LIN {X 0,Y 305.453,Z 160.427,A -85,B 0,C 180,E1 -15811.108,E2 -15811.108} C_VEL
LIN {X 0,Y 305.478,Z 160.428,A -85,B 0,C 180,E1 -15814.08,E2 -15814.08} C_VEL
LIN {X 0,Y 305.457,Z 160.438,A -85,B 0,C 180,E1 -15818.4,E2 -15818.4} C_VEL
LIN {X 0,Y 305.499,Z 160.427,A -85,B 0,C 180,E1 -15821.213,E2 -15821.213} C_VEL
LIN {X 0,Y 305.569,Z 160.419,A -85,B 0,C 180,E1 -15825.346,E2 -15825.346} C_VEL
LIN {X 0,Y 305.622,Z 160.412,A -85,B 0,C 180,E1 -15829.4,E2 -15829.4} C_VEL
LIN {X 0,Y 305.753,Z 160.399,A -85,B 0,C 180,E1 -15832.074,E2 -15832.074} C_VEL
LIN {X 0,Y 305.659,Z 160.409,A -85,B 0,C 180,E1 -15834.724,E2 -15834.724} C_VEL
LIN {X 0,Y 305.938,Z 160.372,A -85,B 0,C 180,E1 -15838.684,E2 -15838.684} C_VEL
LIN {X 0,Y 305.939,Z 160.373,A -85,B 0,C 180,E1 -15841.317,E2 -15841.317} C_VEL
LIN {X 0,Y 305.788,Z 160.391,A -85,B 0,C 180,E1 -15846.599,E2 -15846.599} C_VEL
LIN {X 0,Y 305.699,Z 160.403,A -85,B 0,C 180,E1 -15849.262,E2 -15849.262} C_VEL
LIN {X 0,Y 305.576,Z 160.422,A -85,B 0,C 180,E1 -15853.297,E2 -15853.297} C_VEL
LIN {X 0,Y 305.518,Z 160.424,A -85,B 0,C 180,E1 -15856.025,E2 -15856.025} C_VEL
LIN {X 0,Y 305.483,Z 160.43,A -85,B 0,C 180,E1 -15860.188,E2 -15860.188} C_VEL
LIN {X 0,Y 305.491,Z 160.432,A -85,B 0,C 180,E1 -15863.04,E2 -15863.04} C_VEL
LIN {X 0,Y 305.472,Z 160.431,A -85,B 0,C 180,E1 -15866.197,E2 -15866.197} C_VEL
LIN {X 0,Y 305.451,Z 160.438,A -85,B 0,C 180,E1 -15869.033,E2 -15869.033} C_VEL
LIN {X 0,Y 305.44,Z 160.435,A -85,B 0,C 180,E1 -15871.953,E2 -15871.953} C_VEL
LIN {X 0,Y 305.466,Z 160.436,A -85,B 0,C 180,E1 -15875.114,E2 -15875.114} C_VEL
LIN {X 0,Y 305.437,Z 160.438,A -85,B 0,C 180,E1 -15878.525,E2 -15878.525} C_VEL
LIN {X 0,Y 305.439,Z 160.44,A -85,B 0,C 180,E1 -15882.582,E2 -15882.582} C_VEL
LIN {X 0,Y 305.424,Z 160.441,A -85,B 0,C 180,E1 -15886.344,E2 -15886.344} C_VEL
LIN {X 0,Y 305.414,Z 160.44,A -85,B 0,C 180,E1 -15889.885,E2 -15889.885} C_VEL
LIN {X 0,Y 305.467,Z 160.433,A -85,B 0,C 180,E1 -15893.636,E2 -15893.636} C_VEL
LIN {X 0,Y 305.469,Z 160.437,A -85,B 0,C 180,E1 -15896.483,E2 -15896.483} C_VEL
LIN {X 0,Y 305.467,Z 160.528,A -85,B 0,C 180,E1 -15898.422,E2 -15898.422} C_VEL
LIN {X 0,Y 307.798,Z 171.715,A -85,B 0,C 180,E1 -15901.719,E2 -15901.719} C_VEL
LIN {X 0,Y 309.263,Z 179.963,A -85,B 0,C 180,E1 -15904.058,E2 -15904.058} C_VEL
LIN {X 0,Y 308.728,Z 185.546,A -85,B 0,C 180,E1 -15905.524,E2 -15905.524} C_VEL
LIN {X 0,Y 314.413,Z 227.443,A -85,B 0,C 180,E1 -15906.914,E2 -15906.914} C_VEL
LIN {X 0,Y 312.89,Z 293.878,A -85,B 0,C 180,E1 -15908.462,E2 -15908.462} C_VEL
LIN {X 0,Y 312.195,Z 307.17,A -85,B 0,C 180,E1 -15909.018,E2 -15909.018} C_VEL
LIN {X 0,Y 311.167,Z 320.508,A -85,B 0,C 180,E1 -15909.852,E2 -15909.852} C_VEL
LIN {X 0,Y 310.022,Z 331.7,A -85,B 0,C 180,E1 -15910.809,E2 -15910.809} C_VEL
LIN {X 0,Y 308.738,Z 343.365,A -85,B 0,C 180,E1 -15912.102,E2 -15912.102} C_VEL
LIN {X 0,Y 307.518,Z 354.294,A -85,B 0,C 180,E1 -15913.638,E2 -15913.638} C_VEL
LIN {X 0,Y 306.372,Z 364.129,A -85,B 0,C 180,E1 -15915.384,E2 -15915.384} C_VEL
LIN {X 0,Y 305.291,Z 373.098,A -85,B 0,C 180,E1 -15917.367,E2 -15917.367} C_VEL
LIN {X 0,Y 304.512,Z 380.276,A -85,B 0,C 180,E1 -15919.36,E2 -15919.36} C_VEL
LIN {X 0,Y 304.015,Z 385.985,A -85,B 0,C 180,E1 -15921.358,E2 -15921.358} C_VEL
LIN {X 0,Y 303.748,Z 390.465,A -85,B 0,C 180,E1 -15923.356,E2 -15923.356} C_VEL
LIN {X 0,Y 303.669,Z 392.822,A -85,B 0,C 180,E1 -15924.688,E2 -15924.688} C_VEL
LIN {X 0,Y 303.664,Z 394.742,A -85,B 0,C 180,E1 -15926.018,E2 -15926.018} C_VEL
LIN {X 0,Y 303.642,Z 396.207,A -85,B 0,C 180,E1 -15927.346,E2 -15927.346} C_VEL
LIN {X 0,Y 303.634,Z 397.229,A -85,B 0,C 180,E1 -15928.673,E2 -15928.673} C_VEL
LIN {X 0,Y 303.671,Z 397.858,A -85,B 0,C 180,E1 -15930,E2 -15930} C_VEL
LIN {X 0,Y 303.608,Z 398.092,A -85,B 0,C 180,E1 -15931.326,E2 -15931.326} C_VEL
LIN {X 0,Y 303.622,Z 397.918,A -85,B 0,C 180,E1 -15932.653,E2 -15932.653} C_VEL
LIN {X 0,Y 303.624,Z 397.32,A -85,B 0,C 180,E1 -15933.982,E2 -15933.982} C_VEL
LIN {X 0,Y 303.732,Z 394.961,A -85,B 0,C 180,E1 -15936.643,E2 -15936.643} C_VEL
LIN {X 0,Y 304.114,Z 392.081,A -85,B 0,C 180,E1 -15938.639,E2 -15938.639} C_VEL
LIN {X 0,Y 304.723,Z 388.193,A -85,B 0,C 180,E1 -15940.632,E2 -15940.632} C_VEL
LIN {X 0,Y 305.625,Z 383.199,A -85,B 0,C 180,E1 -15942.618,E2 -15942.618} C_VEL
LIN {X 0,Y 307.01,Z 376.951,A -85,B 0,C 180,E1 -15944.584,E2 -15944.584} C_VEL
LIN {X 0,Y 308.52,Z 369.636,A -85,B 0,C 180,E1 -15946.439,E2 -15946.439} C_VEL
LIN {X 0,Y 310.07,Z 361.462,A -85,B 0,C 180,E1 -15948.125,E2 -15948.125} C_VEL
LIN {X 0,Y 312.018,Z 351.681,A -85,B 0,C 180,E1 -15949.747,E2 -15949.747} C_VEL
LIN {X 0,Y 313.987,Z 341.067,A -85,B 0,C 180,E1 -15951.157,E2 -15951.157} C_VEL
LIN {X 0,Y 315.629,Z 330.837,A -85,B 0,C 180,E1 -15952.243,E2 -15952.243} C_VEL
LIN {X 0,Y 317.331,Z 318.676,A -85,B 0,C 180,E1 -15953.235,E2 -15953.235} C_VEL
LIN {X 0,Y 318.848,Z 305.214,A -85,B 0,C 180,E1 -15954.022,E2 -15954.022} C_VEL
LIN {X 0,Y 319.839,Z 292.7,A -85,B 0,C 180,E1 -15954.504,E2 -15954.504} C_VEL
LIN {X 0,Y 321.622,Z 229.197,A -85,B 0,C 180,E1 -15956.002,E2 -15956.002} C_VEL
LIN {X 0,Y 318.654,Z 211.067,A -85,B 0,C 180,E1 -15956.804,E2 -15956.804} C_VEL
LIN {X 0,Y 314.686,Z 192.542,A -85,B 0,C 180,E1 -15957.753,E2 -15957.753} C_VEL
LIN {X 0,Y 311.096,Z 184.219,A -85,B 0,C 180,E1 -15958.444,E2 -15958.444} C_VEL
LIN {X 0,Y 309.125,Z 174.684,A -85,B 0,C 180,E1 -15961.527,E2 -15961.527} C_VEL
LIN {X 0,Y 306.659,Z 164.84,A -85,B 0,C 180,E1 -15964.956,E2 -15964.956} C_VEL
LIN {X 0,Y 305.47,Z 160.428,A -85,B 0,C 180,E1 -15966.618,E2 -15966.618} C_VEL
LIN {X 0,Y 305.412,Z 160.433,A -85,B 0,C 180,E1 -15970.115,E2 -15970.115} C_VEL
LIN {X 0,Y 305.423,Z 160.439,A -85,B 0,C 180,E1 -15973.656,E2 -15973.656} C_VEL
LIN {X 0,Y 305.436,Z 160.439,A -85,B 0,C 180,E1 -15977.418,E2 -15977.418} C_VEL
LIN {X 0,Y 305.462,Z 160.431,A -85,B 0,C 180,E1 -15981.595,E2 -15981.595} C_VEL
LIN {X 0,Y 305.463,Z 160.429,A -85,B 0,C 180,E1 -15984.886,E2 -15984.886} C_VEL
LIN {X 0,Y 305.443,Z 160.432,A -85,B 0,C 180,E1 -15988.358,E2 -15988.358} C_VEL
LIN {X 0,Y 305.476,Z 160.432,A -85,B 0,C 180,E1 -15991.108,E2 -15991.108} C_VEL
LIN {X 0,Y 305.48,Z 160.424,A -85,B 0,C 180,E1 -15994.079,E2 -15994.079} C_VEL
LIN {X 0,Y 305.457,Z 160.427,A -85,B 0,C 180,E1 -15998.399,E2 -15998.399} C_VEL
LIN {X 0,Y 305.503,Z 160.424,A -85,B 0,C 180,E1 -16001.211,E2 -16001.211} C_VEL
LIN {X 0,Y 305.581,Z 160.419,A -85,B 0,C 180,E1 -16005.345,E2 -16005.345} C_VEL
LIN {X 0,Y 305.625,Z 160.414,A -85,B 0,C 180,E1 -16009.399,E2 -16009.399} C_VEL
LIN {X 0,Y 305.748,Z 160.387,A -85,B 0,C 180,E1 -16012.072,E2 -16012.072} C_VEL
LIN {X 0,Y 305.661,Z 160.407,A -85,B 0,C 180,E1 -16014.722,E2 -16014.722} C_VEL
LIN {X 0,Y 305.947,Z 160.372,A -85,B 0,C 180,E1 -16018.683,E2 -16018.683} C_VEL
LIN {X 0,Y 305.942,Z 160.363,A -85,B 0,C 180,E1 -16021.316,E2 -16021.316} C_VEL
LIN {X 0,Y 305.668,Z 160.401,A -85,B 0,C 180,E1 -16025.276,E2 -16025.276} C_VEL
LIN {X 0,Y 305.748,Z 160.4,A -85,B 0,C 180,E1 -16027.927,E2 -16027.927} C_VEL
LIN {X 0,Y 305.601,Z 160.418,A -85,B 0,C 180,E1 -16031.944,E2 -16031.944} C_VEL
LIN {X 0,Y 305.609,Z 160.409,A -85,B 0,C 180,E1 -16035.014,E2 -16035.014} C_VEL
LIN {X 0,Y 305.547,Z 160.423,A -85,B 0,C 180,E1 -16039.428,E2 -16039.428} C_VEL
LIN {X 0,Y 305.486,Z 160.433,A -85,B 0,C 180,E1 -16043.039,E2 -16043.039} C_VEL
LIN {X 0,Y 305.553,Z 160.425,A -85,B 0,C 180,E1 -16046.229,E2 -16046.229} C_VEL
LIN {X 0,Y 305.495,Z 160.434,A -85,B 0,C 180,E1 -16049.049,E2 -16049.049} C_VEL
LIN {X 0,Y 305.443,Z 160.439,A -85,B 0,C 180,E1 -16051.951,E2 -16051.951} C_VEL
LIN {X 0,Y 305.461,Z 160.436,A -85,B 0,C 180,E1 -16055.112,E2 -16055.112} C_VEL
LIN {X 0,Y 305.481,Z 160.531,A -85,B 0,C 180,E1 -16058.995,E2 -16058.995} C_VEL
LIN {X 0,Y 306.938,Z 166.086,A -85,B 0,C 180,E1 -16061.11,E2 -16061.11} C_VEL
LIN {X 0,Y 315.148,Z 182.086,A -85,B 0,C 180,E1 -16062.566,E2 -16062.566} C_VEL
LIN {X 0,Y 322.647,Z 199.055,A -85,B 0,C 180,E1 -16063.867,E2 -16063.867} C_VEL
LIN {X 0,Y 320.218,Z 273.623,A -85,B 0,C 180,E1 -16065.607,E2 -16065.607} C_VEL
LIN {X 0,Y 319.312,Z 286.842,A -85,B 0,C 180,E1 -16066.168,E2 -16066.168} C_VEL
LIN {X 0,Y 318.139,Z 299.763,A -85,B 0,C 180,E1 -16066.995,E2 -16066.995} C_VEL
LIN {X 0,Y 316.565,Z 311.66,A -85,B 0,C 180,E1 -16068.025,E2 -16068.025} C_VEL
LIN {X 0,Y 314.88,Z 322.44,A -85,B 0,C 180,E1 -16069.228,E2 -16069.228} C_VEL
LIN {X 0,Y 313.124,Z 332.579,A -85,B 0,C 180,E1 -16070.649,E2 -16070.649} C_VEL
LIN {X 0,Y 311.124,Z 342.596,A -85,B 0,C 180,E1 -16072.417,E2 -16072.417} C_VEL
LIN {X 0,Y 309.42,Z 350.599,A -85,B 0,C 180,E1 -16074.178,E2 -16074.178} C_VEL
LIN {X 0,Y 307.952,Z 357.327,A -85,B 0,C 180,E1 -16076.004,E2 -16076.004} C_VEL
LIN {X 0,Y 306.491,Z 363.676,A -85,B 0,C 180,E1 -16078.17,E2 -16078.17} C_VEL
LIN {X 0,Y 305.435,Z 368.51,A -85,B 0,C 180,E1 -16080.349,E2 -16080.349} C_VEL
LIN {X 0,Y 304.584,Z 372.051,A -85,B 0,C 180,E1 -16082.517,E2 -16082.517} C_VEL
LIN {X 0,Y 304.096,Z 374.142,A -85,B 0,C 180,E1 -16084.332,E2 -16084.332} C_VEL
LIN {X 0,Y 303.653,Z 375.725,A -85,B 0,C 180,E1 -16086.83,E2 -16086.83} C_VEL
LIN {X 0,Y 303.54,Z 376.02,A -85,B 0,C 180,E1 -16088.256,E2 -16088.256} C_VEL
LIN {X 0,Y 303.461,Z 375.877,A -85,B 0,C 180,E1 -16089.672,E2 -16089.672} C_VEL
LIN {X 0,Y 303.499,Z 374.866,A -85,B 0,C 180,E1 -16091.696,E2 -16091.696} C_VEL
LIN {X 0,Y 303.653,Z 372.729,A -85,B 0,C 180,E1 -16093.875,E2 -16093.875} C_VEL
LIN {X 0,Y 304.054,Z 369.307,A -85,B 0,C 180,E1 -16096.116,E2 -16096.116} C_VEL
LIN {X 0,Y 304.43,Z 365.405,A -85,B 0,C 180,E1 -16098.008,E2 -16098.008} C_VEL
LIN {X 0,Y 305.114,Z 358.942,A -85,B 0,C 180,E1 -16100.387,E2 -16100.387} C_VEL
LIN {X 0,Y 305.975,Z 351.895,A -85,B 0,C 180,E1 -16102.411,E2 -16102.411} C_VEL
LIN {X 0,Y 306.881,Z 344.682,A -85,B 0,C 180,E1 -16104.085,E2 -16104.085} C_VEL
LIN {X 0,Y 308.05,Z 334.951,A -85,B 0,C 180,E1 -16105.912,E2 -16105.912} C_VEL
LIN {X 0,Y 309.279,Z 325.11,A -85,B 0,C 180,E1 -16107.395,E2 -16107.395} C_VEL
LIN {X 0,Y 310.386,Z 314.381,A -85,B 0,C 180,E1 -16108.703,E2 -16108.703} C_VEL
LIN {X 0,Y 311.427,Z 302.397,A -85,B 0,C 180,E1 -16109.839,E2 -16109.839} C_VEL
LIN {X 0,Y 312.319,Z 289.908,A -85,B 0,C 180,E1 -16110.725,E2 -16110.725} C_VEL
LIN {X 0,Y 312.962,Z 277.052,A -85,B 0,C 180,E1 -16111.367,E2 -16111.367} C_VEL
LIN {X 0,Y 313.42,Z 261.752,A -85,B 0,C 180,E1 -16111.807,E2 -16111.807} C_VEL
LIN {X 0,Y 314.938,Z 194.418,A -85,B 0,C 180,E1 -16113.35,E2 -16113.35} C_VEL
LIN {X 0,Y 312.824,Z 183.531,A -85,B 0,C 180,E1 -16113.751,E2 -16113.751} C_VEL
LIN {X 0,Y 308.878,Z 171.653,A -85,B 0,C 180,E1 -16114.305,E2 -16114.305} C_VEL
LIN {X 0,Y 306.47,Z 164.922,A -85,B 0,C 180,E1 -16114.646,E2 -16114.646} C_VEL
LIN {X 0,Y 305.782,Z 160.401,A -85,B 0,C 180,E1 -16116.102,E2 -16116.102} C_VEL
LIN {X 0,Y 305.689,Z 160.407,A -85,B 0,C 180,E1 -16119.261,E2 -16119.261} C_VEL
LIN {X 0,Y 305.549,Z 160.424,A -85,B 0,C 180,E1 -16123.298,E2 -16123.298} C_VEL
LIN {X 0,Y 305.488,Z 160.432,A -85,B 0,C 180,E1 -16126.026,E2 -16126.026} C_VEL
LIN {X 0,Y 305.475,Z 160.435,A -85,B 0,C 180,E1 -16129.393,E2 -16129.393} C_VEL
LIN {X 0,Y 305.452,Z 160.433,A -85,B 0,C 180,E1 -16133.026,E2 -16133.026} C_VEL
LIN {X 0,Y 305.446,Z 160.426,A -85,B 0,C 180,E1 -16136.19,E2 -16136.19} C_VEL
LIN {X 0,Y 305.421,Z 160.437,A -85,B 0,C 180,E1 -16139.026,E2 -16139.026} C_VEL
LIN {X 0,Y 305.433,Z 160.437,A -85,B 0,C 180,E1 -16141.954,E2 -16141.954} C_VEL
LIN {X 0,Y 305.458,Z 160.435,A -85,B 0,C 180,E1 -16145.114,E2 -16145.114} C_VEL
LIN {X 0,Y 305.43,Z 160.436,A -85,B 0,C 180,E1 -16148.525,E2 -16148.525} C_VEL
LIN {X 0,Y 305.432,Z 160.438,A -85,B 0,C 180,E1 -16152.582,E2 -16152.582} C_VEL
LIN {X 0,Y 305.419,Z 160.433,A -85,B 0,C 180,E1 -16156.345,E2 -16156.345} C_VEL
LIN {X 0,Y 305.422,Z 160.432,A -85,B 0,C 180,E1 -16157.218,E2 -16157.218} C_VEL
LIN {X 0,Y 304.785,Z 160.515,A -85,B 0,C 180,E1 -16158.319,E2 -16158.319} C_VEL
LIN {X 0,Y 301.914,Z 160.873,A -85,B 0,C 180,E1 -16160.112,E2 -16160.112} C_VEL
LIN {X 0,Y 299.485,Z 161.177,A -85,B 0,C 180,E1 -16161.566,E2 -16161.566} C_VEL
LIN {X 0,Y 298.479,Z 161.306,A -85,B 0,C 180,E1 -16162.693,E2 -16162.693} C_VEL
LIN {X 0,Y 298.418,Z 161.311,A -85,B 0,C 180,E1 -16163.075,E2 -16163.075} C_VEL
LIN {X 0,Y 298.407,Z 161.309,A -85,B 0,C 180,E1 -16165.582,E2 -16165.582} C_VEL
LIN {X 0,Y 298.372,Z 161.309,A -85,B 0,C 180,E1 -16168.789,E2 -16168.789} C_VEL
LIN {X 0,Y 298.396,Z 161.304,A -85,B 0,C 180,E1 -16171.898,E2 -16171.898} C_VEL
LIN {X 0,Y 298.413,Z 161.311,A -85,B 0,C 180,E1 -16174.918,E2 -16174.918} C_VEL
LIN {X 0,Y 298.39,Z 161.315,A -85,B 0,C 180,E1 -16177.862,E2 -16177.862} C_VEL
LIN {X 0,Y 298.451,Z 161.306,A -85,B 0,C 180,E1 -16180.752,E2 -16180.752} C_VEL
LIN {X 0,Y 298.512,Z 161.298,A -85,B 0,C 180,E1 -16184.991,E2 -16184.991} C_VEL
LIN {X 0,Y 298.58,Z 161.289,A -85,B 0,C 180,E1 -16189.147,E2 -16189.147} C_VEL
LIN {X 0,Y 298.703,Z 161.275,A -85,B 0,C 180,E1 -16191.885,E2 -16191.885} C_VEL
LIN {X 0,Y 298.63,Z 161.285,A -85,B 0,C 180,E1 -16194.599,E2 -16194.599} C_VEL
LIN {X 0,Y 298.905,Z 161.248,A -85,B 0,C 180,E1 -16198.653,E2 -16198.653} C_VEL
LIN {X 0,Y 298.907,Z 161.249,A -85,B 0,C 180,E1 -16201.348,E2 -16201.348} C_VEL
LIN {X 0,Y 298.737,Z 161.269,A -85,B 0,C 180,E1 -16206.756,E2 -16206.756} C_VEL
LIN {X 0,Y 298.63,Z 161.286,A -85,B 0,C 180,E1 -16209.483,E2 -16209.483} C_VEL
LIN {X 0,Y 298.528,Z 161.3,A -85,B 0,C 180,E1 -16213.617,E2 -16213.617} C_VEL
LIN {X 0,Y 298.458,Z 161.302,A -85,B 0,C 180,E1 -16216.414,E2 -16216.414} C_VEL
LIN {X 0,Y 298.447,Z 161.31,A -85,B 0,C 180,E1 -16219.617,E2 -16219.617} C_VEL
LIN {X 0,Y 298.425,Z 161.312,A -85,B 0,C 180,E1 -16223.601,E2 -16223.601} C_VEL
LIN {X 0,Y 298.411,Z 161.312,A -85,B 0,C 180,E1 -16226.583,E2 -16226.583} C_VEL
LIN {X 0,Y 298.397,Z 161.314,A -85,B 0,C 180,E1 -16229.644,E2 -16229.644} C_VEL
LIN {X 0,Y 298.397,Z 161.316,A -85,B 0,C 180,E1 -16232.801,E2 -16232.801} C_VEL
LIN {X 0,Y 298.445,Z 161.311,A -85,B 0,C 180,E1 -16236.806,E2 -16236.806} C_VEL
LIN {X 0,Y 298.352,Z 161.323,A -85,B 0,C 180,E1 -16241.079,E2 -16241.079} C_VEL
LIN {X 0,Y 298.359,Z 161.321,A -85,B 0,C 180,E1 -16245.035,E2 -16245.035} C_VEL
LIN {X 0,Y 298.352,Z 161.322,A -85,B 0,C 180,E1 -16248.921,E2 -16248.921} C_VEL
LIN {X 0,Y 298.402,Z 161.315,A -85,B 0,C 180,E1 -16252.239,E2 -16252.239} C_VEL
LIN {X 0,Y 298.412,Z 161.313,A -85,B 0,C 180,E1 -16255.581,E2 -16255.581} C_VEL
LIN {X 0,Y 298.445,Z 161.51,A -85,B 0,C 180,E1 -16258.108,E2 -16258.108} C_VEL
LIN {X 0,Y 300.709,Z 172.305,A -85,B 0,C 180,E1 -16261.372,E2 -16261.372} C_VEL
LIN {X 0,Y 302.205,Z 180.572,A -85,B 0,C 180,E1 -16263.777,E2 -16263.777} C_VEL
LIN {X 0,Y 301.998,Z 184.584,A -85,B 0,C 180,E1 -16264.868,E2 -16264.868} C_VEL
LIN {X 0,Y 301.902,Z 185.248,A -85,B 0,C 180,E1 -16265.044,E2 -16265.044} C_VEL
LIN {X 0,Y 307.689,Z 228.186,A -85,B 0,C 180,E1 -16266.518,E2 -16266.518} C_VEL
LIN {X 0,Y 306.092,Z 294.136,A -85,B 0,C 180,E1 -16268.092,E2 -16268.092} C_VEL
LIN {X 0,Y 305.32,Z 308.017,A -85,B 0,C 180,E1 -16268.699,E2 -16268.699} C_VEL
LIN {X 0,Y 304.275,Z 321.004,A -85,B 0,C 180,E1 -16269.552,E2 -16269.552} C_VEL
LIN {X 0,Y 302.985,Z 333.629,A -85,B 0,C 180,E1 -16270.698,E2 -16270.698} C_VEL
LIN {X 0,Y 301.565,Z 344.875,A -85,B 0,C 180,E1 -16272.013,E2 -16272.013} C_VEL
LIN {X 0,Y 300.588,Z 354.013,A -85,B 0,C 180,E1 -16273.357,E2 -16273.357} C_VEL
LIN {X 0,Y 299.481,Z 363.35,A -85,B 0,C 180,E1 -16275.04,E2 -16275.04} C_VEL
LIN {X 0,Y 298.328,Z 372.404,A -85,B 0,C 180,E1 -16277.067,E2 -16277.067} C_VEL
LIN {X 0,Y 297.485,Z 379.68,A -85,B 0,C 180,E1 -16279.105,E2 -16279.105} C_VEL
LIN {X 0,Y 296.97,Z 385.468,A -85,B 0,C 180,E1 -16281.151,E2 -16281.151} C_VEL
LIN {X 0,Y 296.69,Z 390.009,A -85,B 0,C 180,E1 -16283.198,E2 -16283.198} C_VEL
LIN {X 0,Y 296.583,Z 392.393,A -85,B 0,C 180,E1 -16284.561,E2 -16284.561} C_VEL
LIN {X 0,Y 296.579,Z 394.34,A -85,B 0,C 180,E1 -16285.923,E2 -16285.923} C_VEL
LIN {X 0,Y 296.567,Z 395.854,A -85,B 0,C 180,E1 -16287.283,E2 -16287.283} C_VEL
LIN {X 0,Y 296.55,Z 396.906,A -85,B 0,C 180,E1 -16288.642,E2 -16288.642} C_VEL
LIN {X 0,Y 296.582,Z 397.56,A -85,B 0,C 180,E1 -16290,E2 -16290} C_VEL
LIN {X 0,Y 296.525,Z 397.819,A -85,B 0,C 180,E1 -16291.358,E2 -16291.358} C_VEL
LIN {X 0,Y 296.546,Z 397.687,A -85,B 0,C 180,E1 -16292.717,E2 -16292.717} C_VEL
LIN {X 0,Y 296.521,Z 397.121,A -85,B 0,C 180,E1 -16294.077,E2 -16294.077} C_VEL
LIN {X 0,Y 296.657,Z 394.812,A -85,B 0,C 180,E1 -16296.803,E2 -16296.803} C_VEL
LIN {X 0,Y 297.066,Z 391.985,A -85,B 0,C 180,E1 -16298.846,E2 -16298.846} C_VEL
LIN {X 0,Y 297.725,Z 388.151,A -85,B 0,C 180,E1 -16300.885,E2 -16300.885} C_VEL
LIN {X 0,Y 298.668,Z 383.216,A -85,B 0,C 180,E1 -16302.917,E2 -16302.917} C_VEL
LIN {X 0,Y 300.147,Z 377.047,A -85,B 0,C 180,E1 -16304.926,E2 -16304.926} C_VEL
LIN {X 0,Y 301.654,Z 370.06,A -85,B 0,C 180,E1 -16306.767,E2 -16306.767} C_VEL
LIN {X 0,Y 303.376,Z 361.636,A -85,B 0,C 180,E1 -16308.574,E2 -16308.574} C_VEL
LIN {X 0,Y 305.38,Z 352.169,A -85,B 0,C 180,E1 -16310.194,E2 -16310.194} C_VEL
LIN {X 0,Y 307.416,Z 341.709,A -85,B 0,C 180,E1 -16311.632,E2 -16311.632} C_VEL
LIN {X 0,Y 309.39,Z 330.102,A -85,B 0,C 180,E1 -16312.893,E2 -16312.893} C_VEL
LIN {X 0,Y 311.158,Z 317.757,A -85,B 0,C 180,E1 -16313.9,E2 -16313.9} C_VEL
LIN {X 0,Y 312.681,Z 304.814,A -85,B 0,C 180,E1 -16314.659,E2 -16314.659} C_VEL
LIN {X 0,Y 313.678,Z 292.219,A -85,B 0,C 180,E1 -16315.15,E2 -16315.15} C_VEL
LIN {X 0,Y 315.463,Z 229.755,A -85,B 0,C 180,E1 -16316.656,E2 -16316.656} C_VEL
LIN {X 0,Y 312.598,Z 212.284,A -85,B 0,C 180,E1 -16317.456,E2 -16317.456} C_VEL
LIN {X 0,Y 309.058,Z 195.479,A -85,B 0,C 180,E1 -16318.34,E2 -16318.34} C_VEL
LIN {X 0,Y 303.911,Z 183.976,A -85,B 0,C 180,E1 -16319.328,E2 -16319.328} C_VEL
LIN {X 0,Y 302.003,Z 174.977,A -85,B 0,C 180,E1 -16322.36,E2 -16322.36} C_VEL
LIN {X 0,Y 299.515,Z 165.152,A -85,B 0,C 180,E1 -16325.917,E2 -16325.917} C_VEL
LIN {X 0,Y 298.384,Z 161.308,A -85,B 0,C 180,E1 -16327.493,E2 -16327.493} C_VEL
LIN {X 0,Y 298.349,Z 161.309,A -85,B 0,C 180,E1 -16331.268,E2 -16331.268} C_VEL
LIN {X 0,Y 298.357,Z 161.322,A -85,B 0,C 180,E1 -16335.034,E2 -16335.034} C_VEL
LIN {X 0,Y 298.349,Z 161.318,A -85,B 0,C 180,E1 -16338.921,E2 -16338.921} C_VEL
LIN {X 0,Y 298.4,Z 161.309,A -85,B 0,C 180,E1 -16342.239,E2 -16342.239} C_VEL
LIN {X 0,Y 298.41,Z 161.305,A -85,B 0,C 180,E1 -16345.581,E2 -16345.581} C_VEL
LIN {X 0,Y 298.378,Z 161.309,A -85,B 0,C 180,E1 -16348.788,E2 -16348.788} C_VEL
LIN {X 0,Y 298.411,Z 161.311,A -85,B 0,C 180,E1 -16351.898,E2 -16351.898} C_VEL
LIN {X 0,Y 298.422,Z 161.311,A -85,B 0,C 180,E1 -16354.918,E2 -16354.918} C_VEL
LIN {X 0,Y 298.39,Z 161.303,A -85,B 0,C 180,E1 -16357.861,E2 -16357.861} C_VEL
LIN {X 0,Y 298.453,Z 161.303,A -85,B 0,C 180,E1 -16360.75,E2 -16360.75} C_VEL
LIN {X 0,Y 298.512,Z 161.3,A -85,B 0,C 180,E1 -16364.99,E2 -16364.99} C_VEL
LIN {X 0,Y 298.583,Z 161.29,A -85,B 0,C 180,E1 -16369.146,E2 -16369.146} C_VEL
LIN {X 0,Y 298.7,Z 161.265,A -85,B 0,C 180,E1 -16371.884,E2 -16371.884} C_VEL
LIN {X 0,Y 298.631,Z 161.283,A -85,B 0,C 180,E1 -16374.598,E2 -16374.598} C_VEL
LIN {X 0,Y 298.914,Z 161.248,A -85,B 0,C 180,E1 -16378.652,E2 -16378.652} C_VEL
LIN {X 0,Y 298.91,Z 161.239,A -85,B 0,C 180,E1 -16381.347,E2 -16381.347} C_VEL
LIN {X 0,Y 298.637,Z 161.276,A -85,B 0,C 180,E1 -16385.401,E2 -16385.401} C_VEL
LIN {X 0,Y 298.709,Z 161.277,A -85,B 0,C 180,E1 -16388.82,E2 -16388.82} C_VEL
LIN {X 0,Y 298.547,Z 161.291,A -85,B 0,C 180,E1 -16393.615,E2 -16393.615} C_VEL
LIN {X 0,Y 298.488,Z 161.304,A -85,B 0,C 180,E1 -16396.411,E2 -16396.411} C_VEL
LIN {X 0,Y 298.487,Z 161.305,A -85,B 0,C 180,E1 -16399.64,E2 -16399.64} C_VEL
LIN {X 0,Y 298.428,Z 161.314,A -85,B 0,C 180,E1 -16403.599,E2 -16403.599} C_VEL
LIN {X 0,Y 298.491,Z 161.307,A -85,B 0,C 180,E1 -16406.573,E2 -16406.573} C_VEL
LIN {X 0,Y 298.42,Z 161.314,A -85,B 0,C 180,E1 -16409.64,E2 -16409.64} C_VEL
LIN {X 0,Y 298.395,Z 161.314,A -85,B 0,C 180,E1 -16412.799,E2 -16412.799} C_VEL
LIN {X 0,Y 298.449,Z 161.311,A -85,B 0,C 180,E1 -16416.808,E2 -16416.808} C_VEL
LIN {X 0,Y 298.47,Z 161.476,A -85,B 0,C 180,E1 -16418.213,E2 -16418.213} C_VEL
LIN {X 0,Y 299.722,Z 166.368,A -85,B 0,C 180,E1 -16420.152,E2 -16420.152} C_VEL
LIN {X 0,Y 308.004,Z 182.046,A -85,B 0,C 180,E1 -16421.703,E2 -16421.703} C_VEL
LIN {X 0,Y 315.353,Z 198.166,A -85,B 0,C 180,E1 -16423.028,E2 -16423.028} C_VEL
LIN {X 0,Y 316.522,Z 200.984,A -85,B 0,C 180,E1 -16423.238,E2 -16423.238} C_VEL
LIN {X 0,Y 314.088,Z 273.457,A -85,B 0,C 180,E1 -16424.957,E2 -16424.957} C_VEL
LIN {X 0,Y 313.138,Z 286.705,A -85,B 0,C 180,E1 -16425.519,E2 -16425.519} C_VEL
LIN {X 0,Y 311.986,Z 299.331,A -85,B 0,C 180,E1 -16426.332,E2 -16426.332} C_VEL
LIN {X 0,Y 310.547,Z 310.035,A -85,B 0,C 180,E1 -16427.24,E2 -16427.24} C_VEL
LIN {X 0,Y 308.767,Z 321.279,A -85,B 0,C 180,E1 -16428.476,E2 -16428.476} C_VEL
LIN {X 0,Y 306.885,Z 331.563,A -85,B 0,C 180,E1 -16429.902,E2 -16429.902} C_VEL
LIN {X 0,Y 304.885,Z 341.389,A -85,B 0,C 180,E1 -16431.603,E2 -16431.603} C_VEL
LIN {X 0,Y 303.064,Z 349.413,A -85,B 0,C 180,E1 -16433.335,E2 -16433.335} C_VEL
LIN {X 0,Y 301.217,Z 357.516,A -85,B 0,C 180,E1 -16435.542,E2 -16435.542} C_VEL
LIN {X 0,Y 299.786,Z 363.36,A -85,B 0,C 180,E1 -16437.559,E2 -16437.559} C_VEL
LIN {X 0,Y 298.679,Z 368,A -85,B 0,C 180,E1 -16439.609,E2 -16439.609} C_VEL
LIN {X 0,Y 297.716,Z 371.782,A -85,B 0,C 180,E1 -16441.828,E2 -16441.828} C_VEL
LIN {X 0,Y 297.102,Z 374.336,A -85,B 0,C 180,E1 -16444.011,E2 -16444.011} C_VEL
LIN {X 0,Y 296.647,Z 375.855,A -85,B 0,C 180,E1 -16446.25,E2 -16446.25} C_VEL
LIN {X 0,Y 296.476,Z 376.245,A -85,B 0,C 180,E1 -16447.711,E2 -16447.711} C_VEL
LIN {X 0,Y 296.374,Z 376.208,A -85,B 0,C 180,E1 -16449.164,E2 -16449.164} C_VEL
LIN {X 0,Y 296.394,Z 375.193,A -85,B 0,C 180,E1 -16451.523,E2 -16451.523} C_VEL
LIN {X 0,Y 296.499,Z 373.418,A -85,B 0,C 180,E1 -16453.475,E2 -16453.475} C_VEL
LIN {X 0,Y 296.732,Z 371.605,A -85,B 0,C 180,E1 -16454.899,E2 -16454.899} C_VEL
LIN {X 0,Y 297.126,Z 367.969,A -85,B 0,C 180,E1 -16457.015,E2 -16457.015} C_VEL
LIN {X 0,Y 297.615,Z 363.184,A -85,B 0,C 180,E1 -16459.111,E2 -16459.111} C_VEL
LIN {X 0,Y 298.464,Z 356.137,A -85,B 0,C 180,E1 -16461.482,E2 -16461.482} C_VEL
LIN {X 0,Y 299.439,Z 348.108,A -85,B 0,C 180,E1 -16463.599,E2 -16463.599} C_VEL
LIN {X 0,Y 300.499,Z 340.03,A -85,B 0,C 180,E1 -16465.305,E2 -16465.305} C_VEL
LIN {X 0,Y 301.805,Z 330.142,A -85,B 0,C 180,E1 -16466.997,E2 -16466.997} C_VEL
LIN {X 0,Y 303.032,Z 319.461,A -85,B 0,C 180,E1 -16468.468,E2 -16468.468} C_VEL
LIN {X 0,Y 304.183,Z 308.393,A -85,B 0,C 180,E1 -16469.669,E2 -16469.669} C_VEL
LIN {X 0,Y 305.07,Z 296.659,A -85,B 0,C 180,E1 -16470.66,E2 -16470.66} C_VEL
LIN {X 0,Y 305.89,Z 283.321,A -85,B 0,C 180,E1 -16471.481,E2 -16471.481} C_VEL
LIN {X 0,Y 306.471,Z 270.927,A -85,B 0,C 180,E1 -16471.971,E2 -16471.971} C_VEL
LIN {X 0,Y 308.257,Z 195.396,A -85,B 0,C 180,E1 -16473.756,E2 -16473.756} C_VEL
LIN {X 0,Y 306.363,Z 185.693,A -85,B 0,C 180,E1 -16474.124,E2 -16474.124} C_VEL
LIN {X 0,Y 302.811,Z 174.879,A -85,B 0,C 180,E1 -16474.638,E2 -16474.638} C_VEL
LIN {X 0,Y 299.343,Z 165.164,A -85,B 0,C 180,E1 -16475.136,E2 -16475.136} C_VEL
LIN {X 0,Y 298.767,Z 161.273,A -85,B 0,C 180,E1 -16476.416,E2 -16476.416} C_VEL
LIN {X 0,Y 298.62,Z 161.289,A -85,B 0,C 180,E1 -16479.483,E2 -16479.483} C_VEL
LIN {X 0,Y 298.504,Z 161.305,A -85,B 0,C 180,E1 -16483.618,E2 -16483.618} C_VEL
LIN {X 0,Y 298.432,Z 161.31,A -85,B 0,C 180,E1 -16486.416,E2 -16486.416} C_VEL
LIN {X 0,Y 298.421,Z 161.315,A -85,B 0,C 180,E1 -16489.608,E2 -16489.608} C_VEL
LIN {X 0,Y 298.377,Z 161.31,A -85,B 0,C 180,E1 -16493.605,E2 -16493.605} C_VEL
LIN {X 0,Y 298.397,Z 161.303,A -85,B 0,C 180,E1 -16496.584,E2 -16496.584} C_VEL
LIN {X 0,Y 298.354,Z 161.32,A -85,B 0,C 180,E1 -16499.649,E2 -16499.649} C_VEL
LIN {X 0,Y 298.39,Z 161.315,A -85,B 0,C 180,E1 -16502.801,E2 -16502.801} C_VEL
LIN {X 0,Y 298.425,Z 161.306,A -85,B 0,C 180,E1 -16506.803,E2 -16506.803} C_VEL
LIN {X 0,Y 298.371,Z 161.318,A -85,B 0,C 180,E1 -16509.493,E2 -16509.493} C_VEL
LIN {X 0,Y 298.368,Z 161.318,A -85,B 0,C 180,E1 -16513.098,E2 -16513.098} C_VEL
LIN {X 0,Y 298.345,Z 161.313,A -85,B 0,C 180,E1 -16517.2,E2 -16517.2} C_VEL
LIN {X 0,Y 298.383,Z 161.317,A -85,B 0,C 180,E1 -16521.012,E2 -16521.012} C_VEL
LIN {X 0,Y 298.418,Z 161.311,A -85,B 0,C 180,E1 -16523.075,E2 -16523.075} C_VEL
LIN {X 0,Y 297.798,Z 161.391,A -85,B 0,C 180,E1 -16524.201,E2 -16524.201} C_VEL
LIN {X 0,Y 294.926,Z 161.744,A -85,B 0,C 180,E1 -16526.033,E2 -16526.033} C_VEL
LIN {X 0,Y 292.453,Z 162.047,A -85,B 0,C 180,E1 -16527.52,E2 -16527.52} C_VEL
LIN {X 0,Y 291.385,Z 162.179,A -85,B 0,C 180,E1 -16528.673,E2 -16528.673} C_VEL
LIN {X 0,Y 291.297,Z 162.184,A -85,B 0,C 180,E1 -16529.064,E2 -16529.064} C_VEL
LIN {X 0,Y 291.343,Z 162.186,A -85,B 0,C 180,E1 -16533.196,E2 -16533.196} C_VEL
LIN {X 0,Y 291.349,Z 162.191,A -85,B 0,C 180,E1 -16537.298,E2 -16537.298} C_VEL
LIN {X 0,Y 291.386,Z 162.19,A -85,B 0,C 180,E1 -16540.266,E2 -16540.266} C_VEL
LIN {X 0,Y 291.453,Z 162.179,A -85,B 0,C 180,E1 -16544.7,E2 -16544.7} C_VEL
LIN {X 0,Y 291.524,Z 162.168,A -85,B 0,C 180,E1 -16548.881,E2 -16548.881} C_VEL
LIN {X 0,Y 291.657,Z 162.151,A -85,B 0,C 180,E1 -16551.688,E2 -16551.688} C_VEL
LIN {X 0,Y 291.6,Z 162.161,A -85,B 0,C 180,E1 -16554.469,E2 -16554.469} C_VEL
LIN {X 0,Y 291.873,Z 162.124,A -85,B 0,C 180,E1 -16558.621,E2 -16558.621} C_VEL
LIN {X 0,Y 291.874,Z 162.125,A -85,B 0,C 180,E1 -16561.38,E2 -16561.38} C_VEL
LIN {X 0,Y 291.689,Z 162.147,A -85,B 0,C 180,E1 -16566.92,E2 -16566.92} C_VEL
LIN {X 0,Y 291.573,Z 162.167,A -85,B 0,C 180,E1 -16569.715,E2 -16569.715} C_VEL
LIN {X 0,Y 291.487,Z 162.174,A -85,B 0,C 180,E1 -16573.953,E2 -16573.953} C_VEL
LIN {X 0,Y 291.41,Z 162.181,A -85,B 0,C 180,E1 -16576.823,E2 -16576.823} C_VEL
LIN {X 0,Y 291.395,Z 162.186,A -85,B 0,C 180,E1 -16579.842,E2 -16579.842} C_VEL
LIN {X 0,Y 291.363,Z 162.189,A -85,B 0,C 180,E1 -16584.209,E2 -16584.209} C_VEL
LIN {X 0,Y 291.357,Z 162.194,A -85,B 0,C 180,E1 -16587.279,E2 -16587.279} C_VEL
LIN {X 0,Y 291.322,Z 162.195,A -85,B 0,C 180,E1 -16590.439,E2 -16590.439} C_VEL
LIN {X 0,Y 291.348,Z 162.192,A -85,B 0,C 180,E1 -16593.699,E2 -16593.699} C_VEL
LIN {X 0,Y 291.372,Z 162.191,A -85,B 0,C 180,E1 -16597.252,E2 -16597.252} C_VEL
LIN {X 0,Y 291.304,Z 162.201,A -85,B 0,C 180,E1 -16600.648,E2 -16600.648} C_VEL
LIN {X 0,Y 291.286,Z 162.203,A -85,B 0,C 180,E1 -16604.404,E2 -16604.404} C_VEL
LIN {X 0,Y 291.299,Z 162.201,A -85,B 0,C 180,E1 -16608.411,E2 -16608.411} C_VEL
LIN {X 0,Y 291.338,Z 162.193,A -85,B 0,C 180,E1 -16611.155,E2 -16611.155} C_VEL
LIN {X 0,Y 291.359,Z 162.193,A -85,B 0,C 180,E1 -16614.625,E2 -16614.625} C_VEL
LIN {X 0,Y 291.375,Z 162.29,A -85,B 0,C 180,E1 -16617.721,E2 -16617.721} C_VEL
LIN {X 0,Y 293.594,Z 172.853,A -85,B 0,C 180,E1 -16621.004,E2 -16621.004} C_VEL
LIN {X 0,Y 295.303,Z 182.522,A -85,B 0,C 180,E1 -16623.877,E2 -16623.877} C_VEL
LIN {X 0,Y 295.076,Z 185.024,A -85,B 0,C 180,E1 -16624.566,E2 -16624.566} C_VEL
LIN {X 0,Y 300.926,Z 228.389,A -85,B 0,C 180,E1 -16626.088,E2 -16626.088} C_VEL
LIN {X 0,Y 299.367,Z 293.245,A -85,B 0,C 180,E1 -16627.665,E2 -16627.665} C_VEL
LIN {X 0,Y 298.648,Z 306.587,A -85,B 0,C 180,E1 -16628.244,E2 -16628.244} C_VEL
LIN {X 0,Y 297.599,Z 319.381,A -85,B 0,C 180,E1 -16629.072,E2 -16629.072} C_VEL
LIN {X 0,Y 296.392,Z 330.75,A -85,B 0,C 180,E1 -16630.07,E2 -16630.07} C_VEL
LIN {X 0,Y 294.978,Z 342.489,A -85,B 0,C 180,E1 -16631.417,E2 -16631.417} C_VEL
LIN {X 0,Y 293.714,Z 353.063,A -85,B 0,C 180,E1 -16632.955,E2 -16632.955} C_VEL
LIN {X 0,Y 292.595,Z 362.569,A -85,B 0,C 180,E1 -16634.679,E2 -16634.679} C_VEL
LIN {X 0,Y 291.351,Z 371.709,A -85,B 0,C 180,E1 -16636.752,E2 -16636.752} C_VEL
LIN {X 0,Y 290.441,Z 379.063,A -85,B 0,C 180,E1 -16638.838,E2 -16638.838} C_VEL
LIN {X 0,Y 289.909,Z 384.941,A -85,B 0,C 180,E1 -16640.934,E2 -16640.934} C_VEL
LIN {X 0,Y 289.632,Z 389.549,A -85,B 0,C 180,E1 -16643.031,E2 -16643.031} C_VEL
LIN {X 0,Y 289.487,Z 392.065,A -85,B 0,C 180,E1 -16644.494,E2 -16644.494} C_VEL
LIN {X 0,Y 289.478,Z 393.938,A -85,B 0,C 180,E1 -16645.823,E2 -16645.823} C_VEL
LIN {X 0,Y 289.493,Z 395.489,A -85,B 0,C 180,E1 -16647.217,E2 -16647.217} C_VEL
LIN {X 0,Y 289.469,Z 396.583,A -85,B 0,C 180,E1 -16648.609,E2 -16648.609} C_VEL
LIN {X 0,Y 289.497,Z 397.261,A -85,B 0,C 180,E1 -16650,E2 -16650} C_VEL
LIN {X 0,Y 289.471,Z 397.444,A -85,B 0,C 180,E1 -16652.783,E2 -16652.783} C_VEL
LIN {X 0,Y 289.432,Z 396.137,A -85,B 0,C 180,E1 -16655.392,E2 -16655.392} C_VEL
LIN {X 0,Y 289.583,Z 394.665,A -85,B 0,C 180,E1 -16656.97,E2 -16656.97} C_VEL
LIN {X 0,Y 290.036,Z 391.898,A -85,B 0,C 180,E1 -16659.062,E2 -16659.062} C_VEL
LIN {X 0,Y 290.741,Z 388.132,A -85,B 0,C 180,E1 -16661.15,E2 -16661.15} C_VEL
LIN {X 0,Y 291.73,Z 383.274,A -85,B 0,C 180,E1 -16663.23,E2 -16663.23} C_VEL
LIN {X 0,Y 293.299,Z 377.178,A -85,B 0,C 180,E1 -16665.283,E2 -16665.283} C_VEL
LIN {X 0,Y 295.018,Z 369.07,A -85,B 0,C 180,E1 -16667.471,E2 -16667.471} C_VEL
LIN {X 0,Y 297.031,Z 360.229,A -85,B 0,C 180,E1 -16669.345,E2 -16669.345} C_VEL
LIN {X 0,Y 299.218,Z 350.529,A -85,B 0,C 180,E1 -16670.989,E2 -16670.989} C_VEL
LIN {X 0,Y 301.4,Z 339.779,A -85,B 0,C 180,E1 -16672.447,E2 -16672.447} C_VEL
LIN {X 0,Y 303.196,Z 329.342,A -85,B 0,C 180,E1 -16673.569,E2 -16673.569} C_VEL
LIN {X 0,Y 304.884,Z 317.952,A -85,B 0,C 180,E1 -16674.515,E2 -16674.515} C_VEL
LIN {X 0,Y 306.536,Z 304.419,A -85,B 0,C 180,E1 -16675.324,E2 -16675.324} C_VEL
LIN {X 0,Y 307.562,Z 291.643,A -85,B 0,C 180,E1 -16675.825,E2 -16675.825} C_VEL
LIN {X 0,Y 309.373,Z 230.628,A -85,B 0,C 180,E1 -16677.324,E2 -16677.324} C_VEL
LIN {X 0,Y 306.52,Z 213.06,A -85,B 0,C 180,E1 -16678.153,E2 -16678.153} C_VEL
LIN {X 0,Y 303.479,Z 198.524,A -85,B 0,C 180,E1 -16678.951,E2 -16678.951} C_VEL
LIN {X 0,Y 296.724,Z 183.658,A -85,B 0,C 180,E1 -16680.3,E2 -16680.3} C_VEL
LIN {X 0,Y 294.726,Z 174.785,A -85,B 0,C 180,E1 -16683.424,E2 -16683.424} C_VEL
LIN {X 0,Y 292.681,Z 166.905,A -85,B 0,C 180,E1 -16686.4,E2 -16686.4} C_VEL
LIN {X 0,Y 291.332,Z 162.192,A -85,B 0,C 180,E1 -16688.315,E2 -16688.315} C_VEL
LIN {X 0,Y 291.29,Z 162.201,A -85,B 0,C 180,E1 -16692.498,E2 -16692.498} C_VEL
LIN {X 0,Y 291.29,Z 162.198,A -85,B 0,C 180,E1 -16696.37,E2 -16696.37} C_VEL
LIN {X 0,Y 291.358,Z 162.193,A -85,B 0,C 180,E1 -16700.524,E2 -16700.524} C_VEL
LIN {X 0,Y 291.392,Z 162.184,A -85,B 0,C 180,E1 -16702.916,E2 -16702.916} C_VEL
LIN {X 0,Y 291.345,Z 162.187,A -85,B 0,C 180,E1 -16706.301,E2 -16706.301} C_VEL
LIN {X 0,Y 291.366,Z 162.185,A -85,B 0,C 180,E1 -16710.268,E2 -16710.268} C_VEL
LIN {X 0,Y 291.348,Z 162.186,A -85,B 0,C 180,E1 -16714.265,E2 -16714.265} C_VEL
LIN {X 0,Y 291.351,Z 162.179,A -85,B 0,C 180,E1 -16717.296,E2 -16717.296} C_VEL
LIN {X 0,Y 291.386,Z 162.188,A -85,B 0,C 180,E1 -16720.264,E2 -16720.264} C_VEL
LIN {X 0,Y 291.476,Z 162.177,A -85,B 0,C 180,E1 -16724.682,E2 -16724.682} C_VEL
LIN {X 0,Y 291.528,Z 162.169,A -85,B 0,C 180,E1 -16728.88,E2 -16728.88} C_VEL
LIN {X 0,Y 291.653,Z 162.142,A -85,B 0,C 180,E1 -16731.686,E2 -16731.686} C_VEL
LIN {X 0,Y 291.601,Z 162.159,A -85,B 0,C 180,E1 -16734.467,E2 -16734.467} C_VEL
LIN {X 0,Y 291.88,Z 162.124,A -85,B 0,C 180,E1 -16738.62,E2 -16738.62} C_VEL
LIN {X 0,Y 291.878,Z 162.114,A -85,B 0,C 180,E1 -16741.379,E2 -16741.379} C_VEL
LIN {X 0,Y 291.649,Z 162.145,A -85,B 0,C 180,E1 -16746.535,E2 -16746.535} C_VEL
LIN {X 0,Y 291.569,Z 162.157,A -85,B 0,C 180,E1 -16749.713,E2 -16749.713} C_VEL
LIN {X 0,Y 291.516,Z 162.165,A -85,B 0,C 180,E1 -16753.95,E2 -16753.95} C_VEL
LIN {X 0,Y 291.443,Z 162.174,A -85,B 0,C 180,E1 -16758.269,E2 -16758.269} C_VEL
LIN {X 0,Y 291.362,Z 162.187,A -85,B 0,C 180,E1 -16761.211,E2 -16761.211} C_VEL
LIN {X 0,Y 291.383,Z 162.191,A -85,B 0,C 180,E1 -16764.206,E2 -16764.206} C_VEL
LIN {X 0,Y 291.425,Z 162.184,A -85,B 0,C 180,E1 -16767.27,E2 -16767.27} C_VEL
LIN {X 0,Y 291.337,Z 162.193,A -85,B 0,C 180,E1 -16770.436,E2 -16770.436} C_VEL
LIN {X 0,Y 291.343,Z 162.195,A -85,B 0,C 180,E1 -16773.698,E2 -16773.698} C_VEL
LIN {X 0,Y 291.422,Z 162.338,A -85,B 0,C 180,E1 -16777.345,E2 -16777.345} C_VEL
LIN {X 0,Y 292.552,Z 166.684,A -85,B 0,C 180,E1 -16779.142,E2 -16779.142} C_VEL
LIN {X 0,Y 294.7,Z 170.615,A -85,B 0,C 180,E1 -16779.575,E2 -16779.575} C_VEL
LIN {X 0,Y 302.5,Z 185.186,A -85,B 0,C 180,E1 -16781.082,E2 -16781.082} C_VEL
LIN {X 0,Y 309.751,Z 201.145,A -85,B 0,C 180,E1 -16782.453,E2 -16782.453} C_VEL
LIN {X 0,Y 310.49,Z 203.378,A -85,B 0,C 180,E1 -16782.603,E2 -16782.603} C_VEL
LIN {X 0,Y 307.957,Z 273.907,A -85,B 0,C 180,E1 -16784.302,E2 -16784.302} C_VEL
LIN {X 0,Y 306.94,Z 287.519,A -85,B 0,C 180,E1 -16784.897,E2 -16784.897} C_VEL
LIN {X 0,Y 305.714,Z 300.1,A -85,B 0,C 180,E1 -16785.731,E2 -16785.731} C_VEL
LIN {X 0,Y 304.035,Z 311.887,A -85,B 0,C 180,E1 -16786.78,E2 -16786.78} C_VEL
LIN {X 0,Y 302.074,Z 323.436,A -85,B 0,C 180,E1 -16788.115,E2 -16788.115} C_VEL
LIN {X 0,Y 300.01,Z 334.008,A -85,B 0,C 180,E1 -16789.674,E2 -16789.674} C_VEL
LIN {X 0,Y 297.89,Z 343.541,A -85,B 0,C 180,E1 -16791.446,E2 -16791.446} C_VEL
LIN {X 0,Y 295.767,Z 352.552,A -85,B 0,C 180,E1 -16793.555,E2 -16793.555} C_VEL
LIN {X 0,Y 293.883,Z 360.011,A -85,B 0,C 180,E1 -16795.807,E2 -16795.807} C_VEL
LIN {X 0,Y 292.377,Z 365.844,A -85,B 0,C 180,E1 -16798.074,E2 -16798.074} C_VEL
LIN {X 0,Y 291.278,Z 370.182,A -85,B 0,C 180,E1 -16800.296,E2 -16800.296} C_VEL
LIN {X 0,Y 290.372,Z 373.457,A -85,B 0,C 180,E1 -16802.622,E2 -16802.622} C_VEL
LIN {X 0,Y 289.975,Z 374.913,A -85,B 0,C 180,E1 -16804.135,E2 -16804.135} C_VEL
LIN {X 0,Y 289.668,Z 375.911,A -85,B 0,C 180,E1 -16805.641,E2 -16805.641} C_VEL
LIN {X 0,Y 289.432,Z 376.487,A -85,B 0,C 180,E1 -16807.324,E2 -16807.324} C_VEL
LIN {X 0,Y 289.323,Z 376.523,A -85,B 0,C 180,E1 -16808.631,E2 -16808.631} C_VEL
LIN {X 0,Y 289.298,Z 375.521,A -85,B 0,C 180,E1 -16811.338,E2 -16811.338} C_VEL
LIN {X 0,Y 289.375,Z 374.094,A -85,B 0,C 180,E1 -16813.056,E2 -16813.056} C_VEL
LIN {X 0,Y 289.701,Z 371.244,A -85,B 0,C 180,E1 -16815.315,E2 -16815.315} C_VEL
LIN {X 0,Y 290.123,Z 367.546,A -85,B 0,C 180,E1 -16817.408,E2 -16817.408} C_VEL
LIN {X 0,Y 290.633,Z 362.583,A -85,B 0,C 180,E1 -16819.551,E2 -16819.551} C_VEL
LIN {X 0,Y 291.447,Z 356.296,A -85,B 0,C 180,E1 -16821.681,E2 -16821.681} C_VEL
LIN {X 0,Y 292.432,Z 348.474,A -85,B 0,C 180,E1 -16823.792,E2 -16823.792} C_VEL
LIN {X 0,Y 293.513,Z 340.419,A -85,B 0,C 180,E1 -16825.537,E2 -16825.537} C_VEL
LIN {X 0,Y 294.878,Z 330.543,A -85,B 0,C 180,E1 -16827.268,E2 -16827.268} C_VEL
LIN {X 0,Y 296.16,Z 319.6,A -85,B 0,C 180,E1 -16828.81,E2 -16828.81} C_VEL
LIN {X 0,Y 297.321,Z 308.874,A -85,B 0,C 180,E1 -16830,E2 -16830} C_VEL
LIN {X 0,Y 298.241,Z 297.19,A -85,B 0,C 180,E1 -16831.013,E2 -16831.013} C_VEL
LIN {X 0,Y 299.087,Z 283.938,A -85,B 0,C 180,E1 -16831.852,E2 -16831.852} C_VEL
LIN {X 0,Y 299.692,Z 271.861,A -85,B 0,C 180,E1 -16832.352,E2 -16832.352} C_VEL
LIN {X 0,Y 301.556,Z 196.285,A -85,B 0,C 180,E1 -16834.177,E2 -16834.177} C_VEL
LIN {X 0,Y 299.758,Z 187.306,A -85,B 0,C 180,E1 -16834.529,E2 -16834.529} C_VEL
LIN {X 0,Y 295.895,Z 175.881,A -85,B 0,C 180,E1 -16835.095,E2 -16835.095} C_VEL
LIN {X 0,Y 292.22,Z 165.4,A -85,B 0,C 180,E1 -16835.651,E2 -16835.651} C_VEL
LIN {X 0,Y 291.699,Z 162.153,A -85,B 0,C 180,E1 -16836.746,E2 -16836.746} C_VEL
LIN {X 0,Y 291.563,Z 162.168,A -85,B 0,C 180,E1 -16839.714,E2 -16839.714} C_VEL
LIN {X 0,Y 291.467,Z 162.181,A -85,B 0,C 180,E1 -16843.953,E2 -16843.953} C_VEL
LIN {X 0,Y 291.386,Z 162.187,A -85,B 0,C 180,E1 -16846.824,E2 -16846.824} C_VEL
LIN {X 0,Y 291.388,Z 162.189,A -85,B 0,C 180,E1 -16849.843,E2 -16849.843} C_VEL
LIN {X 0,Y 291.321,Z 162.183,A -85,B 0,C 180,E1 -16854.213,E2 -16854.213} C_VEL
LIN {X 0,Y 291.325,Z 162.186,A -85,B 0,C 180,E1 -16857.282,E2 -16857.282} C_VEL
LIN {X 0,Y 291.299,Z 162.196,A -85,B 0,C 180,E1 -16860.442,E2 -16860.442} C_VEL
LIN {X 0,Y 291.341,Z 162.192,A -85,B 0,C 180,E1 -16863.699,E2 -16863.699} C_VEL
LIN {X 0,Y 291.356,Z 162.189,A -85,B 0,C 180,E1 -16867.25,E2 -16867.25} C_VEL
LIN {X 0,Y 291.298,Z 162.199,A -85,B 0,C 180,E1 -16870.649,E2 -16870.649} C_VEL
LIN {X 0,Y 291.28,Z 162.197,A -85,B 0,C 180,E1 -16874.405,E2 -16874.405} C_VEL
LIN {X 0,Y 291.293,Z 162.192,A -85,B 0,C 180,E1 -16878.413,E2 -16878.413} C_VEL
LIN {X 0,Y 291.333,Z 162.194,A -85,B 0,C 180,E1 -16881.156,E2 -16881.156} C_VEL
LIN {X 0,Y 291.355,Z 162.194,A -85,B 0,C 180,E1 -16884.626,E2 -16884.626} C_VEL
LIN {X 0,Y 291.366,Z 162.183,A -85,B 0,C 180,E1 -16887.951,E2 -16887.951} C_VEL
LIN {X 0,Y 291.297,Z 162.184,A -85,B 0,C 180,E1 -16889.064,E2 -16889.064} C_VEL
LIN {X 0,Y 290.635,Z 162.269,A -85,B 0,C 180,E1 -16890.219,E2 -16890.219} C_VEL
LIN {X 0,Y 287.813,Z 162.627,A -85,B 0,C 180,E1 -16892.101,E2 -16892.101} C_VEL
LIN {X 0,Y 285.413,Z 162.929,A -85,B 0,C 180,E1 -16893.628,E2 -16893.628} C_VEL
LIN {X 0,Y 284.372,Z 163.06,A -85,B 0,C 180,E1 -16894.81,E2 -16894.81} C_VEL
LIN {X 0,Y 284.282,Z 163.069,A -85,B 0,C 180,E1 -16895.211,E2 -16895.211} C_VEL
LIN {X 0,Y 284.297,Z 163.073,A -85,B 0,C 180,E1 -16898.235,E2 -16898.235} C_VEL
LIN {X 0,Y 284.312,Z 163.065,A -85,B 0,C 180,E1 -16901.256,E2 -16901.256} C_VEL
LIN {X 0,Y 284.422,Z 163.056,A -85,B 0,C 180,E1 -16904.513,E2 -16904.513} C_VEL
LIN {X 0,Y 284.455,Z 163.05,A -85,B 0,C 180,E1 -16908.601,E2 -16908.601} C_VEL
LIN {X 0,Y 284.613,Z 163.026,A -85,B 0,C 180,E1 -16911.481,E2 -16911.481} C_VEL
LIN {X 0,Y 284.57,Z 163.038,A -85,B 0,C 180,E1 -16914.331,E2 -16914.331} C_VEL
LIN {X 0,Y 284.84,Z 162.999,A -85,B 0,C 180,E1 -16918.587,E2 -16918.587} C_VEL
LIN {X 0,Y 284.841,Z 163.001,A -85,B 0,C 180,E1 -16921.415,E2 -16921.415} C_VEL
LIN {X 0,Y 284.645,Z 163.025,A -85,B 0,C 180,E1 -16927.092,E2 -16927.092} C_VEL
LIN {X 0,Y 284.518,Z 163.044,A -85,B 0,C 180,E1 -16929.958,E2 -16929.958} C_VEL
LIN {X 0,Y 284.423,Z 163.053,A -85,B 0,C 180,E1 -16934.307,E2 -16934.307} C_VEL
LIN {X 0,Y 284.327,Z 163.066,A -85,B 0,C 180,E1 -16938.744,E2 -16938.744} C_VEL
LIN {X 0,Y 284.331,Z 163.07,A -85,B 0,C 180,E1 -16943.297,E2 -16943.297} C_VEL
LIN {X 0,Y 284.333,Z 163.07,A -85,B 0,C 180,E1 -16947.147,E2 -16947.147} C_VEL
LIN {X 0,Y 284.3,Z 163.069,A -85,B 0,C 180,E1 -16950.092,E2 -16950.092} C_VEL
LIN {X 0,Y 284.309,Z 163.072,A -85,B 0,C 180,E1 -16952.946,E2 -16952.946} C_VEL
LIN {X 0,Y 284.331,Z 163.067,A -85,B 0,C 180,E1 -16956.387,E2 -16956.387} C_VEL
LIN {X 0,Y 284.286,Z 163.072,A -85,B 0,C 180,E1 -16959.999,E2 -16959.999} C_VEL
LIN {X 0,Y 284.238,Z 163.079,A -85,B 0,C 180,E1 -16964.188,E2 -16964.188} C_VEL
LIN {X 0,Y 284.244,Z 163.078,A -85,B 0,C 180,E1 -16968.119,E2 -16968.119} C_VEL
LIN {X 0,Y 284.313,Z 163.069,A -85,B 0,C 180,E1 -16972.282,E2 -16972.282} C_VEL
LIN {X 0,Y 284.311,Z 163.071,A -85,B 0,C 180,E1 -16975.35,E2 -16975.35} C_VEL
LIN {X 0,Y 284.296,Z 163.099,A -85,B 0,C 180,E1 -16977.321,E2 -16977.321} C_VEL
LIN {X 0,Y 286.704,Z 174.496,A -85,B 0,C 180,E1 -16980.959,E2 -16980.959} C_VEL
LIN {X 0,Y 288.239,Z 183.087,A -85,B 0,C 180,E1 -16983.577,E2 -16983.577} C_VEL
LIN {X 0,Y 288.249,Z 184.749,A -85,B 0,C 180,E1 -16984.057,E2 -16984.057} C_VEL
LIN {X 0,Y 294.204,Z 229.641,A -85,B 0,C 180,E1 -16985.681,E2 -16985.681} C_VEL
LIN {X 0,Y 292.573,Z 293.454,A -85,B 0,C 180,E1 -16987.271,E2 -16987.271} C_VEL
LIN {X 0,Y 291.798,Z 307.178,A -85,B 0,C 180,E1 -16987.893,E2 -16987.893} C_VEL
LIN {X 0,Y 290.713,Z 319.751,A -85,B 0,C 180,E1 -16988.738,E2 -16988.738} C_VEL
LIN {X 0,Y 289.49,Z 330.951,A -85,B 0,C 180,E1 -16989.76,E2 -16989.76} C_VEL
LIN {X 0,Y 288.037,Z 342.612,A -85,B 0,C 180,E1 -16991.137,E2 -16991.137} C_VEL
LIN {X 0,Y 286.738,Z 353.13,A -85,B 0,C 180,E1 -16992.711,E2 -16992.711} C_VEL
LIN {X 0,Y 285.707,Z 361.723,A -85,B 0,C 180,E1 -16994.301,E2 -16994.301} C_VEL
LIN {X 0,Y 284.624,Z 369.61,A -85,B 0,C 180,E1 -16996.069,E2 -16996.069} C_VEL
LIN {X 0,Y 283.547,Z 377.288,A -85,B 0,C 180,E1 -16998.2,E2 -16998.2} C_VEL
LIN {X 0,Y 282.87,Z 384.383,A -85,B 0,C 180,E1 -17000.706,E2 -17000.706} C_VEL
LIN {X 0,Y 282.567,Z 389.064,A -85,B 0,C 180,E1 -17002.856,E2 -17002.856} C_VEL
LIN {X 0,Y 282.413,Z 391.88,A -85,B 0,C 180,E1 -17004.522,E2 -17004.522} C_VEL
LIN {X 0,Y 282.42,Z 395.11,A -85,B 0,C 180,E1 -17007.147,E2 -17007.147} C_VEL
LIN {X 0,Y 282.39,Z 396.256,A -85,B 0,C 180,E1 -17008.574,E2 -17008.574} C_VEL
LIN {X 0,Y 282.414,Z 396.961,A -85,B 0,C 180,E1 -17010,E2 -17010} C_VEL
LIN {X 0,Y 282.367,Z 397.272,A -85,B 0,C 180,E1 -17011.426,E2 -17011.426} C_VEL
LIN {X 0,Y 282.375,Z 397.196,A -85,B 0,C 180,E1 -17012.853,E2 -17012.853} C_VEL
LIN {X 0,Y 282.345,Z 396.113,A -85,B 0,C 180,E1 -17015.333,E2 -17015.333} C_VEL
LIN {X 0,Y 282.509,Z 394.532,A -85,B 0,C 180,E1 -17017.145,E2 -17017.145} C_VEL
LIN {X 0,Y 282.992,Z 391.825,A -85,B 0,C 180,E1 -17019.289,E2 -17019.289} C_VEL
LIN {X 0,Y 283.744,Z 388.122,A -85,B 0,C 180,E1 -17021.429,E2 -17021.429} C_VEL
LIN {X 0,Y 284.812,Z 383.332,A -85,B 0,C 180,E1 -17023.557,E2 -17023.557} C_VEL
LIN {X 0,Y 286.757,Z 376.191,A -85,B 0,C 180,E1 -17026.005,E2 -17026.005} C_VEL
LIN {X 0,Y 288.552,Z 367.972,A -85,B 0,C 180,E1 -17028.214,E2 -17028.214} C_VEL
LIN {X 0,Y 290.788,Z 358.817,A -85,B 0,C 180,E1 -17030.145,E2 -17030.145} C_VEL
LIN {X 0,Y 293.072,Z 348.89,A -85,B 0,C 180,E1 -17031.82,E2 -17031.82} C_VEL
LIN {X 0,Y 295.406,Z 337.712,A -85,B 0,C 180,E1 -17033.299,E2 -17033.299} C_VEL
LIN {X 0,Y 297.314,Z 326.816,A -85,B 0,C 180,E1 -17034.436,E2 -17034.436} C_VEL
LIN {X 0,Y 299.136,Z 314.794,A -85,B 0,C 180,E1 -17035.39,E2 -17035.39} C_VEL
LIN {X 0,Y 300.614,Z 302.421,A -85,B 0,C 180,E1 -17036.092,E2 -17036.092} C_VEL
LIN {X 0,Y 301.574,Z 289.282,A -85,B 0,C 180,E1 -17036.577,E2 -17036.577} C_VEL
LIN {X 0,Y 303.403,Z 231.916,A -85,B 0,C 180,E1 -17037.999,E2 -17037.999} C_VEL
LIN {X 0,Y 300.678,Z 214.782,A -85,B 0,C 180,E1 -17038.841,E2 -17038.841} C_VEL
LIN {X 0,Y 297.874,Z 201.433,A -85,B 0,C 180,E1 -17039.605,E2 -17039.605} C_VEL
LIN {X 0,Y 291.209,Z 187.044,A -85,B 0,C 180,E1 -17040.973,E2 -17040.973} C_VEL
LIN {X 0,Y 289.472,Z 183.225,A -85,B 0,C 180,E1 -17041.379,E2 -17041.379} C_VEL
LIN {X 0,Y 287.386,Z 174.369,A -85,B 0,C 180,E1 -17044.651,E2 -17044.651} C_VEL
LIN {X 0,Y 285.086,Z 165.904,A -85,B 0,C 180,E1 -17048.047,E2 -17048.047} C_VEL
LIN {X 0,Y 284.306,Z 163.072,A -85,B 0,C 180,E1 -17049.305,E2 -17049.305} C_VEL
LIN {X 0,Y 284.24,Z 163.077,A -85,B 0,C 180,E1 -17053.814,E2 -17053.814} C_VEL
LIN {X 0,Y 284.241,Z 163.08,A -85,B 0,C 180,E1 -17058.118,E2 -17058.118} C_VEL
LIN {X 0,Y 284.31,Z 163.064,A -85,B 0,C 180,E1 -17062.281,E2 -17062.281} C_VEL
LIN {X 0,Y 284.309,Z 163.062,A -85,B 0,C 180,E1 -17065.35,E2 -17065.35} C_VEL
LIN {X 0,Y 284.287,Z 163.064,A -85,B 0,C 180,E1 -17068.724,E2 -17068.724} C_VEL
LIN {X 0,Y 284.276,Z 163.07,A -85,B 0,C 180,E1 -17071.983,E2 -17071.983} C_VEL
LIN {X 0,Y 284.3,Z 163.066,A -85,B 0,C 180,E1 -17076.157,E2 -17076.157} C_VEL
LIN {X 0,Y 284.335,Z 163.067,A -85,B 0,C 180,E1 -17079.927,E2 -17079.927} C_VEL
LIN {X 0,Y 284.416,Z 163.058,A -85,B 0,C 180,E1 -17084.516,E2 -17084.516} C_VEL
LIN {X 0,Y 284.46,Z 163.049,A -85,B 0,C 180,E1 -17088.6,E2 -17088.6} C_VEL
LIN {X 0,Y 284.61,Z 163.02,A -85,B 0,C 180,E1 -17091.479,E2 -17091.479} C_VEL
LIN {X 0,Y 284.571,Z 163.036,A -85,B 0,C 180,E1 -17094.33,E2 -17094.33} C_VEL
LIN {X 0,Y 284.846,Z 163,A -85,B 0,C 180,E1 -17098.585,E2 -17098.585} C_VEL
LIN {X 0,Y 284.845,Z 162.99,A -85,B 0,C 180,E1 -17101.413,E2 -17101.413} C_VEL
LIN {X 0,Y 284.598,Z 163.023,A -85,B 0,C 180,E1 -17106.553,E2 -17106.553} C_VEL
LIN {X 0,Y 284.515,Z 163.034,A -85,B 0,C 180,E1 -17109.956,E2 -17109.956} C_VEL
LIN {X 0,Y 284.464,Z 163.042,A -85,B 0,C 180,E1 -17114.303,E2 -17114.303} C_VEL
LIN {X 0,Y 284.382,Z 163.054,A -85,B 0,C 180,E1 -17118.739,E2 -17118.739} C_VEL
LIN {X 0,Y 284.317,Z 163.062,A -85,B 0,C 180,E1 -17121.763,E2 -17121.763} C_VEL
LIN {X 0,Y 284.34,Z 163.063,A -85,B 0,C 180,E1 -17124.846,E2 -17124.846} C_VEL
LIN {X 0,Y 284.334,Z 163.064,A -85,B 0,C 180,E1 -17128.009,E2 -17128.009} C_VEL
LIN {X 0,Y 284.295,Z 163.072,A -85,B 0,C 180,E1 -17131.273,E2 -17131.273} C_VEL
LIN {X 0,Y 284.34,Z 163.068,A -85,B 0,C 180,E1 -17135.348,E2 -17135.348} C_VEL
LIN {X 0,Y 284.335,Z 163.155,A -85,B 0,C 180,E1 -17136.384,E2 -17136.384} C_VEL
LIN {X 0,Y 285.461,Z 167.211,A -85,B 0,C 180,E1 -17138.086,E2 -17138.086} C_VEL
LIN {X 0,Y 294.461,Z 183.368,A -85,B 0,C 180,E1 -17139.93,E2 -17139.93} C_VEL
LIN {X 0,Y 301.796,Z 198.697,A -85,B 0,C 180,E1 -17141.384,E2 -17141.384} C_VEL
LIN {X 0,Y 304.452,Z 204.924,A -85,B 0,C 180,E1 -17141.907,E2 -17141.907} C_VEL
LIN {X 0,Y 301.874,Z 274.502,A -85,B 0,C 180,E1 -17143.628,E2 -17143.628} C_VEL
LIN {X 0,Y 300.797,Z 288.204,A -85,B 0,C 180,E1 -17144.243,E2 -17144.243} C_VEL
LIN {X 0,Y 299.61,Z 299.966,A -85,B 0,C 180,E1 -17145.037,E2 -17145.037} C_VEL
LIN {X 0,Y 297.827,Z 312.001,A -85,B 0,C 180,E1 -17146.118,E2 -17146.118} C_VEL
LIN {X 0,Y 295.873,Z 323.141,A -85,B 0,C 180,E1 -17147.421,E2 -17147.421} C_VEL
LIN {X 0,Y 293.844,Z 333.04,A -85,B 0,C 180,E1 -17148.873,E2 -17148.873} C_VEL
LIN {X 0,Y 291.538,Z 343.128,A -85,B 0,C 180,E1 -17150.741,E2 -17150.741} C_VEL
LIN {X 0,Y 289.496,Z 351.274,A -85,B 0,C 180,E1 -17152.633,E2 -17152.633} C_VEL
LIN {X 0,Y 287.462,Z 359.125,A -85,B 0,C 180,E1 -17154.933,E2 -17154.933} C_VEL
LIN {X 0,Y 285.796,Z 365.197,A -85,B 0,C 180,E1 -17157.248,E2 -17157.248} C_VEL
LIN {X 0,Y 284.369,Z 370.369,A -85,B 0,C 180,E1 -17159.881,E2 -17159.881} C_VEL
LIN {X 0,Y 283.521,Z 373.229,A -85,B 0,C 180,E1 -17161.902,E2 -17161.902} C_VEL
LIN {X 0,Y 283.056,Z 374.86,A -85,B 0,C 180,E1 -17163.454,E2 -17163.454} C_VEL
LIN {X 0,Y 282.683,Z 375.959,A -85,B 0,C 180,E1 -17164.998,E2 -17164.998} C_VEL
LIN {X 0,Y 282.384,Z 376.743,A -85,B 0,C 180,E1 -17167.05,E2 -17167.05} C_VEL
LIN {X 0,Y 282.188,Z 376.558,A -85,B 0,C 180,E1 -17169.594,E2 -17169.594} C_VEL
LIN {X 0,Y 282.186,Z 375.834,A -85,B 0,C 180,E1 -17171.155,E2 -17171.155} C_VEL
LIN {X 0,Y 282.247,Z 374.744,A -85,B 0,C 180,E1 -17172.614,E2 -17172.614} C_VEL
LIN {X 0,Y 282.523,Z 372.188,A -85,B 0,C 180,E1 -17174.859,E2 -17174.859} C_VEL
LIN {X 0,Y 282.953,Z 368.571,A -85,B 0,C 180,E1 -17177.083,E2 -17177.083} C_VEL
LIN {X 0,Y 283.476,Z 363.808,A -85,B 0,C 180,E1 -17179.284,E2 -17179.284} C_VEL
LIN {X 0,Y 284.331,Z 357.008,A -85,B 0,C 180,E1 -17181.702,E2 -17181.702} C_VEL
LIN {X 0,Y 285.421,Z 348.784,A -85,B 0,C 180,E1 -17183.993,E2 -17183.993} C_VEL
LIN {X 0,Y 286.535,Z 340.739,A -85,B 0,C 180,E1 -17185.78,E2 -17185.78} C_VEL
LIN {X 0,Y 287.872,Z 331.393,A -85,B 0,C 180,E1 -17187.469,E2 -17187.469} C_VEL
LIN {X 0,Y 289.119,Z 321.256,A -85,B 0,C 180,E1 -17188.956,E2 -17188.956} C_VEL
LIN {X 0,Y 290.455,Z 309.257,A -85,B 0,C 180,E1 -17190.347,E2 -17190.347} C_VEL
LIN {X 0,Y 291.407,Z 297.61,A -85,B 0,C 180,E1 -17191.382,E2 -17191.382} C_VEL
LIN {X 0,Y 292.299,Z 284.4,A -85,B 0,C 180,E1 -17192.239,E2 -17192.239} C_VEL
LIN {X 0,Y 292.903,Z 272.503,A -85,B 0,C 180,E1 -17192.751,E2 -17192.751} C_VEL
LIN {X 0,Y 294.834,Z 197.104,A -85,B 0,C 180,E1 -17194.615,E2 -17194.615} C_VEL
LIN {X 0,Y 293.229,Z 189.226,A -85,B 0,C 180,E1 -17194.936,E2 -17194.936} C_VEL
LIN {X 0,Y 289.611,Z 178.588,A -85,B 0,C 180,E1 -17195.483,E2 -17195.483} C_VEL
LIN {X 0,Y 285.135,Z 165.655,A -85,B 0,C 180,E1 -17196.191,E2 -17196.191} C_VEL
LIN {X 0,Y 284.634,Z 163.034,A -85,B 0,C 180,E1 -17197.137,E2 -17197.137} C_VEL
LIN {X 0,Y 284.508,Z 163.047,A -85,B 0,C 180,E1 -17199.958,E2 -17199.958} C_VEL
LIN {X 0,Y 284.401,Z 163.059,A -85,B 0,C 180,E1 -17204.307,E2 -17204.307} C_VEL
LIN {X 0,Y 284.333,Z 163.068,A -85,B 0,C 180,E1 -17207.254,E2 -17207.254} C_VEL
LIN {X 0,Y 284.317,Z 163.068,A -85,B 0,C 180,E1 -17210.247,E2 -17210.247} C_VEL
LIN {X 0,Y 284.288,Z 163.059,A -85,B 0,C 180,E1 -17213.84,E2 -17213.84} C_VEL
LIN {X 0,Y 284.282,Z 163.06,A -85,B 0,C 180,E1 -17217.13,E2 -17217.13} C_VEL
LIN {X 0,Y 284.271,Z 163.072,A -85,B 0,C 180,E1 -17220.085,E2 -17220.085} C_VEL
LIN {X 0,Y 284.302,Z 163.071,A -85,B 0,C 180,E1 -17222.946,E2 -17222.946} C_VEL
LIN {X 0,Y 284.318,Z 163.059,A -85,B 0,C 180,E1 -17226.389,E2 -17226.389} C_VEL
LIN {X 0,Y 284.28,Z 163.071,A -85,B 0,C 180,E1 -17230,E2 -17230} C_VEL
LIN {X 0,Y 284.232,Z 163.074,A -85,B 0,C 180,E1 -17234.189,E2 -17234.189} C_VEL
LIN {X 0,Y 284.238,Z 163.068,A -85,B 0,C 180,E1 -17238.119,E2 -17238.119} C_VEL
LIN {X 0,Y 284.308,Z 163.068,A -85,B 0,C 180,E1 -17242.283,E2 -17242.283} C_VEL
LIN {X 0,Y 284.307,Z 163.066,A -85,B 0,C 180,E1 -17245.352,E2 -17245.352} C_VEL
LIN {X 0,Y 284.265,Z 163.061,A -85,B 0,C 180,E1 -17249.057,E2 -17249.057} C_VEL
LIN {X 0,Y 284.286,Z 163.066,A -85,B 0,C 180,E1 -17252.872,E2 -17252.872} C_VEL
LIN {X 0,Y 284.282,Z 163.069,A -85,B 0,C 180,E1 -17255.211,E2 -17255.211} C_VEL
LIN {X 0,Y 283.599,Z 163.159,A -85,B 0,C 180,E1 -17256.394,E2 -17256.394} C_VEL
LIN {X 0,Y 280.752,Z 163.515,A -85,B 0,C 180,E1 -17258.323,E2 -17258.323} C_VEL
LIN {X 0,Y 278.353,Z 163.811,A -85,B 0,C 180,E1 -17259.889,E2 -17259.889} C_VEL
LIN {X 0,Y 277.332,Z 163.935,A -85,B 0,C 180,E1 -17261.102,E2 -17261.102} C_VEL
LIN {X 0,Y 277.253,Z 163.943,A -85,B 0,C 180,E1 -17261.513,E2 -17261.513} C_VEL
LIN {X 0,Y 277.367,Z 163.932,A -85,B 0,C 180,E1 -17265.323,E2 -17265.323} C_VEL
LIN {X 0,Y 277.454,Z 163.923,A -85,B 0,C 180,E1 -17269.788,E2 -17269.788} C_VEL
LIN {X 0,Y 277.605,Z 163.902,A -85,B 0,C 180,E1 -17272.729,E2 -17272.729} C_VEL
LIN {X 0,Y 277.806,Z 163.875,A -85,B 0,C 180,E1 -17278.551,E2 -17278.551} C_VEL
LIN {X 0,Y 277.808,Z 163.877,A -85,B 0,C 180,E1 -17281.45,E2 -17281.45} C_VEL
LIN {X 0,Y 277.604,Z 163.903,A -85,B 0,C 180,E1 -17287.273,E2 -17287.273} C_VEL
LIN {X 0,Y 277.461,Z 163.921,A -85,B 0,C 180,E1 -17290.214,E2 -17290.214} C_VEL
LIN {X 0,Y 277.376,Z 163.931,A -85,B 0,C 180,E1 -17294.678,E2 -17294.678} C_VEL
LIN {X 0,Y 277.283,Z 163.946,A -85,B 0,C 180,E1 -17299.239,E2 -17299.239} C_VEL
LIN {X 0,Y 277.286,Z 163.943,A -85,B 0,C 180,E1 -17303.925,E2 -17303.925} C_VEL
LIN {X 0,Y 277.273,Z 163.946,A -85,B 0,C 180,E1 -17307.483,E2 -17307.483} C_VEL
LIN {X 0,Y 277.252,Z 163.948,A -85,B 0,C 180,E1 -17310.473,E2 -17310.473} C_VEL
LIN {X 0,Y 277.25,Z 163.948,A -85,B 0,C 180,E1 -17313.896,E2 -17313.896} C_VEL
LIN {X 0,Y 277.264,Z 163.947,A -85,B 0,C 180,E1 -17317.471,E2 -17317.471} C_VEL
LIN {X 0,Y 277.188,Z 163.958,A -85,B 0,C 180,E1 -17321.241,E2 -17321.241} C_VEL
LIN {X 0,Y 277.178,Z 163.959,A -85,B 0,C 180,E1 -17325.232,E2 -17325.232} C_VEL
LIN {X 0,Y 277.188,Z 163.96,A -85,B 0,C 180,E1 -17328.759,E2 -17328.759} C_VEL
LIN {X 0,Y 277.259,Z 163.948,A -85,B 0,C 180,E1 -17332.529,E2 -17332.529} C_VEL
LIN {X 0,Y 277.251,Z 163.953,A -85,B 0,C 180,E1 -17336.104,E2 -17336.104} C_VEL
LIN {X 0,Y 277.283,Z 164.051,A -85,B 0,C 180,E1 -17336.958,E2 -17336.958} C_VEL
LIN {X 0,Y 279.683,Z 175.345,A -85,B 0,C 180,E1 -17340.659,E2 -17340.659} C_VEL
LIN {X 0,Y 281.292,Z 184.481,A -85,B 0,C 180,E1 -17343.518,E2 -17343.518} C_VEL
LIN {X 0,Y 284.942,Z 210.17,A -85,B 0,C 180,E1 -17344.512,E2 -17344.512} C_VEL
LIN {X 0,Y 287.493,Z 230.253,A -85,B 0,C 180,E1 -17345.238,E2 -17345.238} C_VEL
LIN {X 0,Y 285.851,Z 292.99,A -85,B 0,C 180,E1 -17346.835,E2 -17346.835} C_VEL
LIN {X 0,Y 285.094,Z 306.247,A -85,B 0,C 180,E1 -17347.44,E2 -17347.44} C_VEL
LIN {X 0,Y 283.976,Z 319,A -85,B 0,C 180,E1 -17348.304,E2 -17348.304} C_VEL
LIN {X 0,Y 282.595,Z 331.135,A -85,B 0,C 180,E1 -17349.434,E2 -17349.434} C_VEL
LIN {X 0,Y 281.102,Z 342.715,A -85,B 0,C 180,E1 -17350.843,E2 -17350.843} C_VEL
LIN {X 0,Y 279.765,Z 353.169,A -85,B 0,C 180,E1 -17352.455,E2 -17352.455} C_VEL
LIN {X 0,Y 278.781,Z 360.809,A -85,B 0,C 180,E1 -17353.9,E2 -17353.9} C_VEL
LIN {X 0,Y 277.678,Z 368.824,A -85,B 0,C 180,E1 -17355.713,E2 -17355.713} C_VEL
LIN {X 0,Y 276.567,Z 376.623,A -85,B 0,C 180,E1 -17357.898,E2 -17357.898} C_VEL
LIN {X 0,Y 275.847,Z 383.795,A -85,B 0,C 180,E1 -17360.467,E2 -17360.467} C_VEL
LIN {X 0,Y 275.494,Z 388.545,A -85,B 0,C 180,E1 -17362.671,E2 -17362.671} C_VEL
LIN {X 0,Y 275.33,Z 391.707,A -85,B 0,C 180,E1 -17364.571,E2 -17364.571} C_VEL
LIN {X 0,Y 275.347,Z 394.72,A -85,B 0,C 180,E1 -17367.074,E2 -17367.074} C_VEL
LIN {X 0,Y 275.313,Z 395.912,A -85,B 0,C 180,E1 -17368.537,E2 -17368.537} C_VEL
LIN {X 0,Y 275.333,Z 396.658,A -85,B 0,C 180,E1 -17370,E2 -17370} C_VEL
LIN {X 0,Y 275.291,Z 396.997,A -85,B 0,C 180,E1 -17371.463,E2 -17371.463} C_VEL
LIN {X 0,Y 275.281,Z 396.949,A -85,B 0,C 180,E1 -17372.927,E2 -17372.927} C_VEL
LIN {X 0,Y 275.25,Z 396.05,A -85,B 0,C 180,E1 -17375.25,E2 -17375.25} C_VEL
LIN {X 0,Y 275.459,Z 394.399,A -85,B 0,C 180,E1 -17377.329,E2 -17377.329} C_VEL
LIN {X 0,Y 276.206,Z 390.669,A -85,B 0,C 180,E1 -17380.26,E2 -17380.26} C_VEL
LIN {X 0,Y 277.084,Z 386.674,A -85,B 0,C 180,E1 -17382.45,E2 -17382.45} C_VEL
LIN {X 0,Y 278.738,Z 380.58,A -85,B 0,C 180,E1 -17384.977,E2 -17384.977} C_VEL
LIN {X 0,Y 280.477,Z 373.95,A -85,B 0,C 180,E1 -17387.123,E2 -17387.123} C_VEL
LIN {X 0,Y 282.501,Z 365.757,A -85,B 0,C 180,E1 -17389.246,E2 -17389.246} C_VEL
LIN {X 0,Y 284.607,Z 357.404,A -85,B 0,C 180,E1 -17390.981,E2 -17390.981} C_VEL
LIN {X 0,Y 287.077,Z 347.144,A -85,B 0,C 180,E1 -17392.68,E2 -17392.68} C_VEL
LIN {X 0,Y 289.427,Z 335.653,A -85,B 0,C 180,E1 -17394.19,E2 -17394.19} C_VEL
LIN {X 0,Y 291.505,Z 324.345,A -85,B 0,C 180,E1 -17395.337,E2 -17395.337} C_VEL
LIN {X 0,Y 293.311,Z 312.741,A -85,B 0,C 180,E1 -17396.217,E2 -17396.217} C_VEL
LIN {X 0,Y 294.851,Z 299.495,A -85,B 0,C 180,E1 -17396.928,E2 -17396.928} C_VEL
LIN {X 0,Y 295.713,Z 285.997,A -85,B 0,C 180,E1 -17397.393,E2 -17397.393} C_VEL
LIN {X 0,Y 297.421,Z 232.482,A -85,B 0,C 180,E1 -17398.744,E2 -17398.744} C_VEL
LIN {X 0,Y 294.508,Z 214.456,A -85,B 0,C 180,E1 -17399.672,E2 -17399.672} C_VEL
LIN {X 0,Y 292.229,Z 204.038,A -85,B 0,C 180,E1 -17400.304,E2 -17400.304} C_VEL
LIN {X 0,Y 286.037,Z 190.751,A -85,B 0,C 180,E1 -17401.622,E2 -17401.622} C_VEL
LIN {X 0,Y 282.26,Z 182.915,A -85,B 0,C 180,E1 -17402.483,E2 -17402.483} C_VEL
LIN {X 0,Y 279.748,Z 172.693,A -85,B 0,C 180,E1 -17406.493,E2 -17406.493} C_VEL
LIN {X 0,Y 277.221,Z 163.942,A -85,B 0,C 180,E1 -17410.281,E2 -17410.281} C_VEL
LIN {X 0,Y 277.193,Z 163.959,A -85,B 0,C 180,E1 -17413.201,E2 -17413.201} C_VEL
LIN {X 0,Y 277.194,Z 163.956,A -85,B 0,C 180,E1 -17417.33,E2 -17417.33} C_VEL
LIN {X 0,Y 277.254,Z 163.943,A -85,B 0,C 180,E1 -17421.795,E2 -17421.795} C_VEL
LIN {X 0,Y 277.28,Z 163.945,A -85,B 0,C 180,E1 -17424.34,E2 -17424.34} C_VEL
LIN {X 0,Y 277.242,Z 163.949,A -85,B 0,C 180,E1 -17427.835,E2 -17427.835} C_VEL
LIN {X 0,Y 277.237,Z 163.949,A -85,B 0,C 180,E1 -17431.206,E2 -17431.206} C_VEL
LIN {X 0,Y 277.237,Z 163.945,A -85,B 0,C 180,E1 -17434.471,E2 -17434.471} C_VEL
LIN {X 0,Y 277.249,Z 163.935,A -85,B 0,C 180,E1 -17437.651,E2 -17437.651} C_VEL
LIN {X 0,Y 277.278,Z 163.941,A -85,B 0,C 180,E1 -17440.761,E2 -17440.761} C_VEL
LIN {X 0,Y 277.383,Z 163.932,A -85,B 0,C 180,E1 -17445.322,E2 -17445.322} C_VEL
LIN {X 0,Y 277.455,Z 163.924,A -85,B 0,C 180,E1 -17449.786,E2 -17449.786} C_VEL
LIN {X 0,Y 277.603,Z 163.895,A -85,B 0,C 180,E1 -17452.727,E2 -17452.727} C_VEL
LIN {X 0,Y 277.812,Z 163.877,A -85,B 0,C 180,E1 -17458.55,E2 -17458.55} C_VEL
LIN {X 0,Y 277.812,Z 163.866,A -85,B 0,C 180,E1 -17461.449,E2 -17461.449} C_VEL
LIN {X 0,Y 277.552,Z 163.9,A -85,B 0,C 180,E1 -17466.566,E2 -17466.566} C_VEL
LIN {X 0,Y 277.561,Z 163.907,A -85,B 0,C 180,E1 -17469.068,E2 -17469.068} C_VEL
LIN {X 0,Y 277.41,Z 163.928,A -85,B 0,C 180,E1 -17473.179,E2 -17473.179} C_VEL
LIN {X 0,Y 277.363,Z 163.935,A -85,B 0,C 180,E1 -17476.183,E2 -17476.183} C_VEL
LIN {X 0,Y 277.337,Z 163.94,A -85,B 0,C 180,E1 -17480.345,E2 -17480.345} C_VEL
LIN {X 0,Y 277.292,Z 163.946,A -85,B 0,C 180,E1 -17484.157,E2 -17484.157} C_VEL
LIN {X 0,Y 277.327,Z 163.938,A -85,B 0,C 180,E1 -17487.505,E2 -17487.505} C_VEL
LIN {X 0,Y 277.271,Z 163.945,A -85,B 0,C 180,E1 -17490.481,E2 -17490.481} C_VEL
LIN {X 0,Y 277.319,Z 163.942,A -85,B 0,C 180,E1 -17495.318,E2 -17495.318} C_VEL
LIN {X 0,Y 278.289,Z 167.501,A -85,B 0,C 180,E1 -17496.914,E2 -17496.914} C_VEL
LIN {X 0,Y 280.571,Z 171.445,A -85,B 0,C 180,E1 -17497.43,E2 -17497.43} C_VEL
LIN {X 0,Y 289.285,Z 187.029,A -85,B 0,C 180,E1 -17499.296,E2 -17499.296} C_VEL
LIN {X 0,Y 296.279,Z 201.714,A -85,B 0,C 180,E1 -17500.737,E2 -17500.737} C_VEL
LIN {X 0,Y 298.539,Z 207.02,A -85,B 0,C 180,E1 -17501.2,E2 -17501.2} C_VEL
LIN {X 0,Y 295.925,Z 274.244,A -85,B 0,C 180,E1 -17502.881,E2 -17502.881} C_VEL
LIN {X 0,Y 294.843,Z 287.501,A -85,B 0,C 180,E1 -17503.471,E2 -17503.471} C_VEL
LIN {X 0,Y 293.537,Z 300.187,A -85,B 0,C 180,E1 -17504.334,E2 -17504.334} C_VEL
LIN {X 0,Y 291.657,Z 312.199,A -85,B 0,C 180,E1 -17505.427,E2 -17505.427} C_VEL
LIN {X 0,Y 289.449,Z 324.17,A -85,B 0,C 180,E1 -17506.864,E2 -17506.864} C_VEL
LIN {X 0,Y 287.243,Z 334.353,A -85,B 0,C 180,E1 -17508.42,E2 -17508.42} C_VEL
LIN {X 0,Y 285.082,Z 343.319,A -85,B 0,C 180,E1 -17510.136,E2 -17510.136} C_VEL
LIN {X 0,Y 282.967,Z 351.247,A -85,B 0,C 180,E1 -17512.002,E2 -17512.002} C_VEL
LIN {X 0,Y 281.099,Z 358.128,A -85,B 0,C 180,E1 -17514.017,E2 -17514.017} C_VEL
LIN {X 0,Y 279.276,Z 364.526,A -85,B 0,C 180,E1 -17516.383,E2 -17516.383} C_VEL
LIN {X 0,Y 277.86,Z 369.416,A -85,B 0,C 180,E1 -17518.768,E2 -17518.768} C_VEL
LIN {X 0,Y 276.727,Z 372.997,A -85,B 0,C 180,E1 -17521.149,E2 -17521.149} C_VEL
LIN {X 0,Y 276.122,Z 374.957,A -85,B 0,C 180,E1 -17522.977,E2 -17522.977} C_VEL
LIN {X 0,Y 275.734,Z 375.998,A -85,B 0,C 180,E1 -17524.323,E2 -17524.323} C_VEL
LIN {X 0,Y 275.315,Z 377.001,A -85,B 0,C 180,E1 -17526.775,E2 -17526.775} C_VEL
LIN {X 0,Y 275.129,Z 376.95,A -85,B 0,C 180,E1 -17529.046,E2 -17529.046} C_VEL
LIN {X 0,Y 275.109,Z 376.157,A -85,B 0,C 180,E1 -17530.943,E2 -17530.943} C_VEL
LIN {X 0,Y 275.261,Z 373.871,A -85,B 0,C 180,E1 -17533.689,E2 -17533.689} C_VEL
LIN {X 0,Y 275.581,Z 371.194,A -85,B 0,C 180,E1 -17535.714,E2 -17535.714} C_VEL
LIN {X 0,Y 276.097,Z 366.632,A -85,B 0,C 180,E1 -17538.25,E2 -17538.25} C_VEL
LIN {X 0,Y 276.911,Z 360.204,A -85,B 0,C 180,E1 -17540.873,E2 -17540.873} C_VEL
LIN {X 0,Y 277.853,Z 353.207,A -85,B 0,C 180,E1 -17543.1,E2 -17543.1} C_VEL
LIN {X 0,Y 278.876,Z 346.047,A -85,B 0,C 180,E1 -17544.94,E2 -17544.94} C_VEL
LIN {X 0,Y 280.103,Z 337.391,A -85,B 0,C 180,E1 -17546.764,E2 -17546.764} C_VEL
LIN {X 0,Y 281.483,Z 327.543,A -85,B 0,C 180,E1 -17548.435,E2 -17548.435} C_VEL
LIN {X 0,Y 282.881,Z 316,A -85,B 0,C 180,E1 -17550,E2 -17550} C_VEL
LIN {X 0,Y 284.085,Z 304.228,A -85,B 0,C 180,E1 -17551.241,E2 -17551.241} C_VEL
LIN {X 0,Y 285.1,Z 291.977,A -85,B 0,C 180,E1 -17552.208,E2 -17552.208} C_VEL
LIN {X 0,Y 285.848,Z 278.705,A -85,B 0,C 180,E1 -17552.951,E2 -17552.951} C_VEL
LIN {X 0,Y 286.365,Z 265.6,A -85,B 0,C 180,E1 -17553.386,E2 -17553.386} C_VEL
LIN {X 0,Y 288.1,Z 197.761,A -85,B 0,C 180,E1 -17555.08,E2 -17555.08} C_VEL
LIN {X 0,Y 286.64,Z 190.792,A -85,B 0,C 180,E1 -17555.376,E2 -17555.376} C_VEL
LIN {X 0,Y 278.003,Z 165.905,A -85,B 0,C 180,E1 -17556.761,E2 -17556.761} C_VEL
LIN {X 0,Y 277.587,Z 163.913,A -85,B 0,C 180,E1 -17557.547,E2 -17557.547} C_VEL
LIN {X 0,Y 277.447,Z 163.926,A -85,B 0,C 180,E1 -17560.214,E2 -17560.214} C_VEL
LIN {X 0,Y 277.36,Z 163.935,A -85,B 0,C 180,E1 -17564.679,E2 -17564.679} C_VEL
LIN {X 0,Y 277.268,Z 163.947,A -85,B 0,C 180,E1 -17569.24,E2 -17569.24} C_VEL
LIN {X 0,Y 277.251,Z 163.934,A -85,B 0,C 180,E1 -17573.928,E2 -17573.928} C_VEL
LIN {X 0,Y 277.232,Z 163.94,A -85,B 0,C 180,E1 -17577.469,E2 -17577.469} C_VEL
LIN {X 0,Y 277.225,Z 163.949,A -85,B 0,C 180,E1 -17580.466,E2 -17580.466} C_VEL
LIN {X 0,Y 277.243,Z 163.946,A -85,B 0,C 180,E1 -17583.897,E2 -17583.897} C_VEL
LIN {X 0,Y 277.252,Z 163.946,A -85,B 0,C 180,E1 -17587.472,E2 -17587.472} C_VEL
LIN {X 0,Y 277.182,Z 163.959,A -85,B 0,C 180,E1 -17591.242,E2 -17591.242} C_VEL
LIN {X 0,Y 277.172,Z 163.949,A -85,B 0,C 180,E1 -17595.233,E2 -17595.233} C_VEL
LIN {X 0,Y 277.182,Z 163.95,A -85,B 0,C 180,E1 -17598.76,E2 -17598.76} C_VEL
LIN {X 0,Y 277.254,Z 163.948,A -85,B 0,C 180,E1 -17602.53,E2 -17602.53} C_VEL
LIN {X 0,Y 277.246,Z 163.946,A -85,B 0,C 180,E1 -17606.105,E2 -17606.105} C_VEL
LIN {X 0,Y 277.228,Z 163.934,A -85,B 0,C 180,E1 -17609.536,E2 -17609.536} C_VEL
LIN {X 0,Y 277.251,Z 163.942,A -85,B 0,C 180,E1 -17612.854,E2 -17612.854} C_VEL
LIN {X 0,Y 277.256,Z 163.946,A -85,B 0,C 180,E1 -17616.074,E2 -17616.074} C_VEL
LIN {X 0,Y 277.274,Z 163.943,A -85,B 0,C 180,E1 -17620.762,E2 -17620.762} C_VEL
LIN {X 0,Y 277.253,Z 163.943,A -85,B 0,C 180,E1 -17621.513,E2 -17621.513} C_VEL
LIN {X 0,Y 276.591,Z 164.028,A -85,B 0,C 180,E1 -17622.725,E2 -17622.725} C_VEL
LIN {X 0,Y 273.739,Z 164.385,A -85,B 0,C 180,E1 -17624.702,E2 -17624.702} C_VEL
LIN {X 0,Y 271.357,Z 164.685,A -85,B 0,C 180,E1 -17626.309,E2 -17626.309} C_VEL
LIN {X 0,Y 270.394,Z 164.803,A -85,B 0,C 180,E1 -17627.553,E2 -17627.553} C_VEL
LIN {X 0,Y 270.347,Z 164.811,A -85,B 0,C 180,E1 -17627.975,E2 -17627.975} C_VEL
LIN {X 0,Y 270.531,Z 164.779,A -85,B 0,C 180,E1 -17631.033,E2 -17631.033} C_VEL
LIN {X 0,Y 270.512,Z 164.791,A -85,B 0,C 180,E1 -17634.036,E2 -17634.036} C_VEL
LIN {X 0,Y 270.772,Z 164.752,A -85,B 0,C 180,E1 -17638.514,E2 -17638.514} C_VEL
LIN {X 0,Y 270.773,Z 164.754,A -85,B 0,C 180,E1 -17641.488,E2 -17641.488} C_VEL
LIN {X 0,Y 270.566,Z 164.78,A -85,B 0,C 180,E1 -17647.463,E2 -17647.463} C_VEL
LIN {X 0,Y 270.413,Z 164.799,A -85,B 0,C 180,E1 -17650.483,E2 -17650.483} C_VEL
LIN {X 0,Y 270.343,Z 164.808,A -85,B 0,C 180,E1 -17655.069,E2 -17655.069} C_VEL
LIN {X 0,Y 270.225,Z 164.824,A -85,B 0,C 180,E1 -17659.762,E2 -17659.762} C_VEL
LIN {X 0,Y 270.228,Z 164.823,A -85,B 0,C 180,E1 -17664.591,E2 -17664.591} C_VEL
LIN {X 0,Y 270.202,Z 164.825,A -85,B 0,C 180,E1 -17667.917,E2 -17667.917} C_VEL
LIN {X 0,Y 270.178,Z 164.831,A -85,B 0,C 180,E1 -17671.35,E2 -17671.35} C_VEL
LIN {X 0,Y 270.203,Z 164.83,A -85,B 0,C 180,E1 -17674.906,E2 -17674.906} C_VEL
LIN {X 0,Y 270.202,Z 164.83,A -85,B 0,C 180,E1 -17678.711,E2 -17678.711} C_VEL
LIN {X 0,Y 270.152,Z 164.835,A -85,B 0,C 180,E1 -17683.245,E2 -17683.245} C_VEL
LIN {X 0,Y 270.155,Z 164.833,A -85,B 0,C 180,E1 -17687.438,E2 -17687.438} C_VEL
LIN {X 0,Y 270.211,Z 164.824,A -85,B 0,C 180,E1 -17691.374,E2 -17691.374} C_VEL
LIN {X 0,Y 270.202,Z 164.828,A -85,B 0,C 180,E1 -17695.094,E2 -17695.094} C_VEL
LIN {X 0,Y 270.236,Z 164.913,A -85,B 0,C 180,E1 -17696.544,E2 -17696.544} C_VEL
LIN {X 0,Y 272.828,Z 177.268,A -85,B 0,C 180,E1 -17700.696,E2 -17700.696} C_VEL
LIN {X 0,Y 274.111,Z 184.387,A -85,B 0,C 180,E1 -17702.953,E2 -17702.953} C_VEL
LIN {X 0,Y 275.508,Z 190.193,A -85,B 0,C 180,E1 -17703.232,E2 -17703.232} C_VEL
LIN {X 0,Y 280.789,Z 231.19,A -85,B 0,C 180,E1 -17704.781,E2 -17704.781} C_VEL
LIN {X 0,Y 279.115,Z 292.856,A -85,B 0,C 180,E1 -17706.389,E2 -17706.389} C_VEL
LIN {X 0,Y 278.327,Z 306.069,A -85,B 0,C 180,E1 -17707.008,E2 -17707.008} C_VEL
LIN {X 0,Y 277.202,Z 318.225,A -85,B 0,C 180,E1 -17707.843,E2 -17707.843} C_VEL
LIN {X 0,Y 275.966,Z 329.723,A -85,B 0,C 180,E1 -17708.917,E2 -17708.917} C_VEL
LIN {X 0,Y 274.332,Z 341.509,A -85,B 0,C 180,E1 -17710.351,E2 -17710.351} C_VEL
LIN {X 0,Y 272.982,Z 352.136,A -85,B 0,C 180,E1 -17712.004,E2 -17712.004} C_VEL
LIN {X 0,Y 271.888,Z 359.895,A -85,B 0,C 180,E1 -17713.48,E2 -17713.48} C_VEL
LIN {X 0,Y 270.717,Z 368.018,A -85,B 0,C 180,E1 -17715.338,E2 -17715.338} C_VEL
LIN {X 0,Y 269.587,Z 375.956,A -85,B 0,C 180,E1 -17717.58,E2 -17717.58} C_VEL
LIN {X 0,Y 268.981,Z 381.343,A -85,B 0,C 180,E1 -17719.461,E2 -17719.461} C_VEL
LIN {X 0,Y 268.502,Z 386.576,A -85,B 0,C 180,E1 -17721.723,E2 -17721.723} C_VEL
LIN {X 0,Y 268.252,Z 390.615,A -85,B 0,C 180,E1 -17723.984,E2 -17723.984} C_VEL
LIN {X 0,Y 268.202,Z 392.687,A -85,B 0,C 180,E1 -17725.491,E2 -17725.491} C_VEL
LIN {X 0,Y 268.252,Z 394.329,A -85,B 0,C 180,E1 -17726.996,E2 -17726.996} C_VEL
LIN {X 0,Y 268.239,Z 395.554,A -85,B 0,C 180,E1 -17728.498,E2 -17728.498} C_VEL
LIN {X 0,Y 268.254,Z 396.355,A -85,B 0,C 180,E1 -17730,E2 -17730} C_VEL
LIN {X 0,Y 268.215,Z 396.722,A -85,B 0,C 180,E1 -17731.501,E2 -17731.501} C_VEL
LIN {X 0,Y 268.19,Z 396.702,A -85,B 0,C 180,E1 -17733.004,E2 -17733.004} C_VEL
LIN {X 0,Y 268.224,Z 395.498,A -85,B 0,C 180,E1 -17736.016,E2 -17736.016} C_VEL
LIN {X 0,Y 268.729,Z 392.635,A -85,B 0,C 180,E1 -17739.028,E2 -17739.028} C_VEL
LIN {X 0,Y 269.461,Z 389.391,A -85,B 0,C 180,E1 -17741.28,E2 -17741.28} C_VEL
LIN {X 0,Y 270.493,Z 385.106,A -85,B 0,C 180,E1 -17743.523,E2 -17743.523} C_VEL
LIN {X 0,Y 272.475,Z 378.651,A -85,B 0,C 180,E1 -17746.098,E2 -17746.098} C_VEL
LIN {X 0,Y 274.03,Z 372.902,A -85,B 0,C 180,E1 -17747.924,E2 -17747.924} C_VEL
LIN {X 0,Y 275.816,Z 366.05,A -85,B 0,C 180,E1 -17749.732,E2 -17749.732} C_VEL
LIN {X 0,Y 278.004,Z 357.826,A -85,B 0,C 180,E1 -17751.504,E2 -17751.504} C_VEL
LIN {X 0,Y 280.576,Z 347.802,A -85,B 0,C 180,E1 -17753.236,E2 -17753.236} C_VEL
LIN {X 0,Y 283.012,Z 336.51,A -85,B 0,C 180,E1 -17754.775,E2 -17754.775} C_VEL
LIN {X 0,Y 285.174,Z 325.468,A -85,B 0,C 180,E1 -17755.941,E2 -17755.941} C_VEL
LIN {X 0,Y 287.19,Z 313.214,A -85,B 0,C 180,E1 -17756.919,E2 -17756.919} C_VEL
LIN {X 0,Y 288.804,Z 300.164,A -85,B 0,C 180,E1 -17757.644,E2 -17757.644} C_VEL
LIN {X 0,Y 289.739,Z 286.499,A -85,B 0,C 180,E1 -17758.139,E2 -17758.139} C_VEL
LIN {X 0,Y 291.54,Z 233.576,A -85,B 0,C 180,E1 -17759.499,E2 -17759.499} C_VEL
LIN {X 0,Y 288.561,Z 215.05,A -85,B 0,C 180,E1 -17760.487,E2 -17760.487} C_VEL
LIN {X 0,Y 286.891,Z 207.256,A -85,B 0,C 180,E1 -17760.973,E2 -17760.973} C_VEL
LIN {X 0,Y 279.536,Z 191.492,A -85,B 0,C 180,E1 -17762.621,E2 -17762.621} C_VEL
LIN {X 0,Y 276.84,Z 186.395,A -85,B 0,C 180,E1 -17763.24,E2 -17763.24} C_VEL
LIN {X 0,Y 274.957,Z 182.507,A -85,B 0,C 180,E1 -17763.733,E2 -17763.733} C_VEL
LIN {X 0,Y 272.923,Z 174.448,A -85,B 0,C 180,E1 -17767.033,E2 -17767.033} C_VEL
LIN {X 0,Y 270.693,Z 166.742,A -85,B 0,C 180,E1 -17770.472,E2 -17770.472} C_VEL
LIN {X 0,Y 270.152,Z 164.821,A -85,B 0,C 180,E1 -17771.413,E2 -17771.413} C_VEL
LIN {X 0,Y 270.131,Z 164.839,A -85,B 0,C 180,E1 -17775.374,E2 -17775.374} C_VEL
LIN {X 0,Y 270.149,Z 164.829,A -85,B 0,C 180,E1 -17779.429,E2 -17779.429} C_VEL
LIN {X 0,Y 270.211,Z 164.825,A -85,B 0,C 180,E1 -17783.257,E2 -17783.257} C_VEL
LIN {X 0,Y 270.204,Z 164.826,A -85,B 0,C 180,E1 -17786.892,E2 -17786.892} C_VEL
LIN {X 0,Y 270.183,Z 164.824,A -85,B 0,C 180,E1 -17790.38,E2 -17790.38} C_VEL
LIN {X 0,Y 270.183,Z 164.818,A -85,B 0,C 180,E1 -17793.755,E2 -17793.755} C_VEL
LIN {X 0,Y 270.184,Z 164.816,A -85,B 0,C 180,E1 -17797.034,E2 -17797.034} C_VEL
LIN {X 0,Y 270.221,Z 164.824,A -85,B 0,C 180,E1 -17800.238,E2 -17800.238} C_VEL
LIN {X 0,Y 270.345,Z 164.809,A -85,B 0,C 180,E1 -17804.931,E2 -17804.931} C_VEL
LIN {X 0,Y 270.387,Z 164.804,A -85,B 0,C 180,E1 -17809.516,E2 -17809.516} C_VEL
LIN {X 0,Y 270.564,Z 164.77,A -85,B 0,C 180,E1 -17812.537,E2 -17812.537} C_VEL
LIN {X 0,Y 270.777,Z 164.753,A -85,B 0,C 180,E1 -17818.512,E2 -17818.512} C_VEL
LIN {X 0,Y 270.779,Z 164.741,A -85,B 0,C 180,E1 -17821.486,E2 -17821.486} C_VEL
LIN {X 0,Y 270.564,Z 164.778,A -85,B 0,C 180,E1 -17827.462,E2 -17827.462} C_VEL
LIN {X 0,Y 270.411,Z 164.789,A -85,B 0,C 180,E1 -17830.481,E2 -17830.481} C_VEL
LIN {X 0,Y 270.378,Z 164.797,A -85,B 0,C 180,E1 -17835.065,E2 -17835.065} C_VEL
LIN {X 0,Y 270.29,Z 164.817,A -85,B 0,C 180,E1 -17839.755,E2 -17839.755} C_VEL
LIN {X 0,Y 270.238,Z 164.821,A -85,B 0,C 180,E1 -17844.588,E2 -17844.588} C_VEL
LIN {X 0,Y 270.272,Z 164.816,A -85,B 0,C 180,E1 -17847.908,E2 -17847.908} C_VEL
LIN {X 0,Y 270.183,Z 164.83,A -85,B 0,C 180,E1 -17851.347,E2 -17851.347} C_VEL
LIN {X 0,Y 270.251,Z 164.976,A -85,B 0,C 180,E1 -17854.328,E2 -17854.328} C_VEL
LIN {X 0,Y 271.016,Z 167.749,A -85,B 0,C 180,E1 -17855.637,E2 -17855.637} C_VEL
LIN {X 0,Y 273.379,Z 171.688,A -85,B 0,C 180,E1 -17856.202,E2 -17856.202} C_VEL
LIN {X 0,Y 281.018,Z 184.892,A -85,B 0,C 180,E1 -17857.95,E2 -17857.95} C_VEL
LIN {X 0,Y 287.585,Z 197.71,A -85,B 0,C 180,E1 -17859.38,E2 -17859.38} C_VEL
LIN {X 0,Y 292.662,Z 209.357,A -85,B 0,C 180,E1 -17860.469,E2 -17860.469} C_VEL
LIN {X 0,Y 289.956,Z 274.896,A -85,B 0,C 180,E1 -17862.137,E2 -17862.137} C_VEL
LIN {X 0,Y 288.776,Z 288.824,A -85,B 0,C 180,E1 -17862.784,E2 -17862.784} C_VEL
LIN {X 0,Y 287.324,Z 301.561,A -85,B 0,C 180,E1 -17863.689,E2 -17863.689} C_VEL
LIN {X 0,Y 285.541,Z 312.455,A -85,B 0,C 180,E1 -17864.708,E2 -17864.708} C_VEL
LIN {X 0,Y 283.454,Z 323.412,A -85,B 0,C 180,E1 -17866.034,E2 -17866.034} C_VEL
LIN {X 0,Y 281.192,Z 333.471,A -85,B 0,C 180,E1 -17867.559,E2 -17867.559} C_VEL
LIN {X 0,Y 279.134,Z 341.73,A -85,B 0,C 180,E1 -17869.109,E2 -17869.109} C_VEL
LIN {X 0,Y 276.812,Z 350.236,A -85,B 0,C 180,E1 -17871.07,E2 -17871.07} C_VEL
LIN {X 0,Y 274.456,Z 358.356,A -85,B 0,C 180,E1 -17873.461,E2 -17873.461} C_VEL
LIN {X 0,Y 272.765,Z 363.92,A -85,B 0,C 180,E1 -17875.537,E2 -17875.537} C_VEL
LIN {X 0,Y 271.217,Z 368.91,A -85,B 0,C 180,E1 -17877.913,E2 -17877.913} C_VEL
LIN {X 0,Y 269.966,Z 372.732,A -85,B 0,C 180,E1 -17880.355,E2 -17880.355} C_VEL
LIN {X 0,Y 269.121,Z 375.178,A -85,B 0,C 180,E1 -17882.608,E2 -17882.608} C_VEL
LIN {X 0,Y 268.46,Z 376.879,A -85,B 0,C 180,E1 -17885.237,E2 -17885.237} C_VEL
LIN {X 0,Y 268.226,Z 377.292,A -85,B 0,C 180,E1 -17886.857,E2 -17886.857} C_VEL
LIN {X 0,Y 268.05,Z 377.27,A -85,B 0,C 180,E1 -17888.465,E2 -17888.465} C_VEL
LIN {X 0,Y 268.016,Z 376.474,A -85,B 0,C 180,E1 -17890.732,E2 -17890.732} C_VEL
LIN {X 0,Y 268.107,Z 374.536,A -85,B 0,C 180,E1 -17893.241,E2 -17893.241} C_VEL
LIN {X 0,Y 268.475,Z 371.651,A -85,B 0,C 180,E1 -17895.592,E2 -17895.592} C_VEL
LIN {X 0,Y 268.924,Z 367.67,A -85,B 0,C 180,E1 -17897.932,E2 -17897.932} C_VEL
LIN {X 0,Y 269.57,Z 362.522,A -85,B 0,C 180,E1 -17900.244,E2 -17900.244} C_VEL
LIN {X 0,Y 270.484,Z 356.031,A -85,B 0,C 180,E1 -17902.536,E2 -17902.536} C_VEL
LIN {X 0,Y 271.663,Z 347.877,A -85,B 0,C 180,E1 -17904.805,E2 -17904.805} C_VEL
LIN {X 0,Y 272.849,Z 339.562,A -85,B 0,C 180,E1 -17906.678,E2 -17906.678} C_VEL
LIN {X 0,Y 274.414,Z 329.346,A -85,B 0,C 180,E1 -17908.533,E2 -17908.533} C_VEL
LIN {X 0,Y 275.655,Z 319.261,A -85,B 0,C 180,E1 -17910,E2 -17910} C_VEL
LIN {X 0,Y 276.937,Z 308.239,A -85,B 0,C 180,E1 -17911.273,E2 -17911.273} C_VEL
LIN {X 0,Y 278.022,Z 296.136,A -85,B 0,C 180,E1 -17912.355,E2 -17912.355} C_VEL
LIN {X 0,Y 278.856,Z 283.763,A -85,B 0,C 180,E1 -17913.161,E2 -17913.161} C_VEL
LIN {X 0,Y 279.523,Z 270.898,A -85,B 0,C 180,E1 -17913.694,E2 -17913.694} C_VEL
LIN {X 0,Y 281.461,Z 198.634,A -85,B 0,C 180,E1 -17915.555,E2 -17915.555} C_VEL
LIN {X 0,Y 279.868,Z 191.735,A -85,B 0,C 180,E1 -17915.87,E2 -17915.87} C_VEL
LIN {X 0,Y 270.805,Z 166.187,A -85,B 0,C 180,E1 -17917.343,E2 -17917.343} C_VEL
LIN {X 0,Y 270.551,Z 164.787,A -85,B 0,C 180,E1 -17917.917,E2 -17917.917} C_VEL
LIN {X 0,Y 270.342,Z 164.812,A -85,B 0,C 180,E1 -17922.004,E2 -17922.004} C_VEL
LIN {X 0,Y 270.312,Z 164.816,A -85,B 0,C 180,E1 -17925.852,E2 -17925.852} C_VEL
LIN {X 0,Y 270.237,Z 164.821,A -85,B 0,C 180,E1 -17930.572,E2 -17930.572} C_VEL
LIN {X 0,Y 270.173,Z 164.812,A -85,B 0,C 180,E1 -17934.596,E2 -17934.596} C_VEL
LIN {X 0,Y 270.181,Z 164.822,A -85,B 0,C 180,E1 -17937.919,E2 -17937.919} C_VEL
LIN {X 0,Y 270.166,Z 164.834,A -85,B 0,C 180,E1 -17941.351,E2 -17941.351} C_VEL
LIN {X 0,Y 270.195,Z 164.825,A -85,B 0,C 180,E1 -17944.907,E2 -17944.907} C_VEL
LIN {X 0,Y 270.196,Z 164.824,A -85,B 0,C 180,E1 -17948.711,E2 -17948.711} C_VEL
LIN {X 0,Y 270.146,Z 164.831,A -85,B 0,C 180,E1 -17953.246,E2 -17953.246} C_VEL
LIN {X 0,Y 270.149,Z 164.822,A -85,B 0,C 180,E1 -17957.439,E2 -17957.439} C_VEL
LIN {X 0,Y 270.207,Z 164.824,A -85,B 0,C 180,E1 -17961.375,E2 -17961.375} C_VEL
LIN {X 0,Y 270.198,Z 164.824,A -85,B 0,C 180,E1 -17965.095,E2 -17965.095} C_VEL
LIN {X 0,Y 270.171,Z 164.813,A -85,B 0,C 180,E1 -17969.142,E2 -17969.142} C_VEL
LIN {X 0,Y 270.188,Z 164.813,A -85,B 0,C 180,E1 -17972.178,E2 -17972.178} C_VEL
LIN {X 0,Y 270.183,Z 164.825,A -85,B 0,C 180,E1 -17975.565,E2 -17975.565} C_VEL
LIN {X 0,Y 270.219,Z 164.826,A -85,B 0,C 180,E1 -17980.239,E2 -17980.239} C_VEL
LIN {X 0,Y 270.338,Z 164.808,A -85,B 0,C 180,E1 -17984.933,E2 -17984.933} C_VEL
LIN {X 0,Y 270.347,Z 164.811,A -85,B 0,C 180,E1 -17987.975,E2 -17987.975} C_VEL
LIN {X 0,Y 269.786,Z 164.888,A -85,B 0,C 180,E1 -17989.221,E2 -17989.221} C_VEL
LIN {X 0,Y 267.039,Z 165.23,A -85,B 0,C 180,E1 -17991.253,E2 -17991.253} C_VEL
LIN {X 0,Y 263.768,Z 165.628,A -85,B 0,C 180,E1 -17993.753,E2 -17993.753} C_VEL
LIN {X 0,Y 263.39,Z 165.673,A -85,B 0,C 180,E1 -17994.618,E2 -17994.618} C_VEL
LIN {X 0,Y 263.735,Z 165.628,A -85,B 0,C 180,E1 -17998.474,E2 -17998.474} C_VEL
LIN {X 0,Y 263.737,Z 165.63,A -85,B 0,C 180,E1 -18001.528,E2 -18001.528} C_VEL
LIN {X 0,Y 263.53,Z 165.655,A -85,B 0,C 180,E1 -18007.664,E2 -18007.664} C_VEL
LIN {X 0,Y 263.352,Z 165.678,A -85,B 0,C 180,E1 -18010.767,E2 -18010.767} C_VEL
LIN {X 0,Y 263.292,Z 165.685,A -85,B 0,C 180,E1 -18015.482,E2 -18015.482} C_VEL
LIN {X 0,Y 263.212,Z 165.696,A -85,B 0,C 180,E1 -18020.312,E2 -18020.312} C_VEL
LIN {X 0,Y 263.171,Z 165.704,A -85,B 0,C 180,E1 -18025.296,E2 -18025.296} C_VEL
LIN {X 0,Y 263.138,Z 165.707,A -85,B 0,C 180,E1 -18028.735,E2 -18028.735} C_VEL
LIN {X 0,Y 263.132,Z 165.706,A -85,B 0,C 180,E1 -18032.289,E2 -18032.289} C_VEL
LIN {X 0,Y 263.183,Z 165.704,A -85,B 0,C 180,E1 -18036.762,E2 -18036.762} C_VEL
LIN {X 0,Y 263.096,Z 165.713,A -85,B 0,C 180,E1 -18039.875,E2 -18039.875} C_VEL
LIN {X 0,Y 263.08,Z 165.715,A -85,B 0,C 180,E1 -18043.994,E2 -18043.994} C_VEL
LIN {X 0,Y 263.112,Z 165.712,A -85,B 0,C 180,E1 -18048.411,E2 -18048.411} C_VEL
LIN {X 0,Y 263.161,Z 165.703,A -85,B 0,C 180,E1 -18052.103,E2 -18052.103} C_VEL
LIN {X 0,Y 263.169,Z 165.739,A -85,B 0,C 180,E1 -18056.101,E2 -18056.101} C_VEL
LIN {X 0,Y 265.411,Z 176.36,A -85,B 0,C 180,E1 -18059.793,E2 -18059.793} C_VEL
LIN {X 0,Y 266.843,Z 183.901,A -85,B 0,C 180,E1 -18062.301,E2 -18062.301} C_VEL
LIN {X 0,Y 268.887,Z 191.012,A -85,B 0,C 180,E1 -18062.708,E2 -18062.708} C_VEL
LIN {X 0,Y 274.128,Z 232.163,A -85,B 0,C 180,E1 -18064.305,E2 -18064.305} C_VEL
LIN {X 0,Y 272.392,Z 292.72,A -85,B 0,C 180,E1 -18065.922,E2 -18065.922} C_VEL
LIN {X 0,Y 271.522,Z 306.656,A -85,B 0,C 180,E1 -18066.599,E2 -18066.599} C_VEL
LIN {X 0,Y 270.368,Z 318.596,A -85,B 0,C 180,E1 -18067.454,E2 -18067.454} C_VEL
LIN {X 0,Y 269.074,Z 329.914,A -85,B 0,C 180,E1 -18068.551,E2 -18068.551} C_VEL
LIN {X 0,Y 267.418,Z 341.613,A -85,B 0,C 180,E1 -18070.022,E2 -18070.022} C_VEL
LIN {X 0,Y 265.998,Z 352.349,A -85,B 0,C 180,E1 -18071.746,E2 -18071.746} C_VEL
LIN {X 0,Y 264.787,Z 360.793,A -85,B 0,C 180,E1 -18073.421,E2 -18073.421} C_VEL
LIN {X 0,Y 263.614,Z 368.716,A -85,B 0,C 180,E1 -18075.328,E2 -18075.328} C_VEL
LIN {X 0,Y 262.428,Z 376.42,A -85,B 0,C 180,E1 -18077.628,E2 -18077.628} C_VEL
LIN {X 0,Y 261.748,Z 382.614,A -85,B 0,C 180,E1 -18079.949,E2 -18079.949} C_VEL
LIN {X 0,Y 261.338,Z 387.507,A -85,B 0,C 180,E1 -18082.272,E2 -18082.272} C_VEL
LIN {X 0,Y 261.134,Z 391.46,A -85,B 0,C 180,E1 -18084.75,E2 -18084.75} C_VEL
LIN {X 0,Y 261.161,Z 393.938,A -85,B 0,C 180,E1 -18086.914,E2 -18086.914} C_VEL
LIN {X 0,Y 261.165,Z 395.194,A -85,B 0,C 180,E1 -18088.458,E2 -18088.458} C_VEL
LIN {X 0,Y 261.177,Z 396.043,A -85,B 0,C 180,E1 -18090,E2 -18090} C_VEL
LIN {X 0,Y 261.141,Z 396.448,A -85,B 0,C 180,E1 -18091.542,E2 -18091.542} C_VEL
LIN {X 0,Y 261.101,Z 396.455,A -85,B 0,C 180,E1 -18093.086,E2 -18093.086} C_VEL
LIN {X 0,Y 261.149,Z 395.318,A -85,B 0,C 180,E1 -18096.179,E2 -18096.179} C_VEL
LIN {X 0,Y 261.33,Z 394.133,A -85,B 0,C 180,E1 -18097.728,E2 -18097.728} C_VEL
LIN {X 0,Y 262.184,Z 390.528,A -85,B 0,C 180,E1 -18100.815,E2 -18100.815} C_VEL
LIN {X 0,Y 263.162,Z 386.671,A -85,B 0,C 180,E1 -18103.12,E2 -18103.12} C_VEL
LIN {X 0,Y 264.714,Z 381.718,A -85,B 0,C 180,E1 -18105.396,E2 -18105.396} C_VEL
LIN {X 0,Y 266.615,Z 375.523,A -85,B 0,C 180,E1 -18107.646,E2 -18107.646} C_VEL
LIN {X 0,Y 268.69,Z 367.857,A -85,B 0,C 180,E1 -18109.879,E2 -18109.879} C_VEL
LIN {X 0,Y 271.44,Z 358.267,A -85,B 0,C 180,E1 -18112.051,E2 -18112.051} C_VEL
LIN {X 0,Y 274.111,Z 348.404,A -85,B 0,C 180,E1 -18113.817,E2 -18113.817} C_VEL
LIN {X 0,Y 276.629,Z 337.367,A -85,B 0,C 180,E1 -18115.386,E2 -18115.386} C_VEL
LIN {X 0,Y 279.186,Z 324.843,A -85,B 0,C 180,E1 -18116.742,E2 -18116.742} C_VEL
LIN {X 0,Y 281.273,Z 312.437,A -85,B 0,C 180,E1 -18117.734,E2 -18117.734} C_VEL
LIN {X 0,Y 282.896,Z 299.751,A -85,B 0,C 180,E1 -18118.442,E2 -18118.442} C_VEL
LIN {X 0,Y 283.846,Z 286.469,A -85,B 0,C 180,E1 -18118.929,E2 -18118.929} C_VEL
LIN {X 0,Y 285.774,Z 235.147,A -85,B 0,C 180,E1 -18120.26,E2 -18120.26} C_VEL
LIN {X 0,Y 282.958,Z 217.287,A -85,B 0,C 180,E1 -18121.24,E2 -18121.24} C_VEL
LIN {X 0,Y 281.536,Z 210.521,A -85,B 0,C 180,E1 -18121.675,E2 -18121.675} C_VEL
LIN {X 0,Y 275.965,Z 198.316,A -85,B 0,C 180,E1 -18122.984,E2 -18122.984} C_VEL
LIN {X 0,Y 271.826,Z 190.159,A -85,B 0,C 180,E1 -18123.978,E2 -18123.978} C_VEL
LIN {X 0,Y 269.599,Z 186.083,A -85,B 0,C 180,E1 -18124.521,E2 -18124.521} C_VEL
LIN {X 0,Y 267.69,Z 182.154,A -85,B 0,C 180,E1 -18125.047,E2 -18125.047} C_VEL
LIN {X 0,Y 265.484,Z 173.857,A -85,B 0,C 180,E1 -18128.654,E2 -18128.654} C_VEL
LIN {X 0,Y 263.112,Z 165.71,A -85,B 0,C 180,E1 -18132.602,E2 -18132.602} C_VEL
LIN {X 0,Y 263.081,Z 165.712,A -85,B 0,C 180,E1 -18136.161,E2 -18136.161} C_VEL
LIN {X 0,Y 263.093,Z 165.712,A -85,B 0,C 180,E1 -18140.124,E2 -18140.124} C_VEL
LIN {X 0,Y 263.16,Z 165.705,A -85,B 0,C 180,E1 -18144.017,E2 -18144.017} C_VEL
LIN {X 0,Y 263.13,Z 165.707,A -85,B 0,C 180,E1 -18147.711,E2 -18147.711} C_VEL
LIN {X 0,Y 263.143,Z 165.703,A -85,B 0,C 180,E1 -18151.807,E2 -18151.807} C_VEL
LIN {X 0,Y 263.118,Z 165.701,A -85,B 0,C 180,E1 -18156.38,E2 -18156.38} C_VEL
LIN {X 0,Y 263.209,Z 165.698,A -85,B 0,C 180,E1 -18159.688,E2 -18159.688} C_VEL
LIN {X 0,Y 263.292,Z 165.689,A -85,B 0,C 180,E1 -18164.518,E2 -18164.518} C_VEL
LIN {X 0,Y 263.332,Z 165.682,A -85,B 0,C 180,E1 -18169.232,E2 -18169.232} C_VEL
LIN {X 0,Y 263.528,Z 165.645,A -85,B 0,C 180,E1 -18172.336,E2 -18172.336} C_VEL
LIN {X 0,Y 263.74,Z 165.63,A -85,B 0,C 180,E1 -18178.472,E2 -18178.472} C_VEL
LIN {X 0,Y 263.744,Z 165.617,A -85,B 0,C 180,E1 -18181.526,E2 -18181.526} C_VEL
LIN {X 0,Y 263.528,Z 165.657,A -85,B 0,C 180,E1 -18187.662,E2 -18187.662} C_VEL
LIN {X 0,Y 263.353,Z 165.669,A -85,B 0,C 180,E1 -18190.766,E2 -18190.766} C_VEL
LIN {X 0,Y 263.324,Z 165.678,A -85,B 0,C 180,E1 -18195.479,E2 -18195.479} C_VEL
LIN {X 0,Y 263.256,Z 165.695,A -85,B 0,C 180,E1 -18200.306,E2 -18200.306} C_VEL
LIN {X 0,Y 263.193,Z 165.697,A -85,B 0,C 180,E1 -18205.292,E2 -18205.292} C_VEL
LIN {X 0,Y 263.179,Z 165.701,A -85,B 0,C 180,E1 -18208.729,E2 -18208.729} C_VEL
LIN {X 0,Y 263.158,Z 165.705,A -85,B 0,C 180,E1 -18213.079,E2 -18213.079} C_VEL
LIN {X 0,Y 263.873,Z 168.186,A -85,B 0,C 180,E1 -18214.295,E2 -18214.295} C_VEL
LIN {X 0,Y 266.007,Z 171.764,A -85,B 0,C 180,E1 -18214.843,E2 -18214.843} C_VEL
LIN {X 0,Y 272.061,Z 181.631,A -85,B 0,C 180,E1 -18216.315,E2 -18216.315} C_VEL
LIN {X 0,Y 280.077,Z 196.424,A -85,B 0,C 180,E1 -18218.179,E2 -18218.179} C_VEL
LIN {X 0,Y 286.812,Z 211.143,A -85,B 0,C 180,E1 -18219.688,E2 -18219.688} C_VEL
LIN {X 0,Y 284.111,Z 274.753,A -85,B 0,C 180,E1 -18221.334,E2 -18221.334} C_VEL
LIN {X 0,Y 282.921,Z 287.94,A -85,B 0,C 180,E1 -18221.933,E2 -18221.933} C_VEL
LIN {X 0,Y 281.505,Z 300.685,A -85,B 0,C 180,E1 -18222.83,E2 -18222.83} C_VEL
LIN {X 0,Y 279.472,Z 312.707,A -85,B 0,C 180,E1 -18223.958,E2 -18223.958} C_VEL
LIN {X 0,Y 277.202,Z 324.092,A -85,B 0,C 180,E1 -18225.364,E2 -18225.364} C_VEL
LIN {X 0,Y 274.648,Z 334.86,A -85,B 0,C 180,E1 -18227.054,E2 -18227.054} C_VEL
LIN {X 0,Y 272.213,Z 344.018,A -85,B 0,C 180,E1 -18228.879,E2 -18228.879} C_VEL
LIN {X 0,Y 269.882,Z 351.958,A -85,B 0,C 180,E1 -18230.839,E2 -18230.839} C_VEL
LIN {X 0,Y 267.466,Z 359.815,A -85,B 0,C 180,E1 -18233.289,E2 -18233.289} C_VEL
LIN {X 0,Y 265.62,Z 365.514,A -85,B 0,C 180,E1 -18235.582,E2 -18235.582} C_VEL
LIN {X 0,Y 264.138,Z 369.901,A -85,B 0,C 180,E1 -18237.849,E2 -18237.849} C_VEL
LIN {X 0,Y 262.867,Z 373.492,A -85,B 0,C 180,E1 -18240.356,E2 -18240.356} C_VEL
LIN {X 0,Y 261.939,Z 375.921,A -85,B 0,C 180,E1 -18242.863,E2 -18242.863} C_VEL
LIN {X 0,Y 261.499,Z 376.932,A -85,B 0,C 180,E1 -18244.532,E2 -18244.532} C_VEL
LIN {X 0,Y 261.213,Z 377.506,A -85,B 0,C 180,E1 -18246.198,E2 -18246.198} C_VEL
LIN {X 0,Y 261,Z 377.586,A -85,B 0,C 180,E1 -18247.853,E2 -18247.853} C_VEL
LIN {X 0,Y 260.915,Z 376.788,A -85,B 0,C 180,E1 -18250.517,E2 -18250.517} C_VEL
LIN {X 0,Y 260.962,Z 375.201,A -85,B 0,C 180,E1 -18252.768,E2 -18252.768} C_VEL
LIN {X 0,Y 261.36,Z 372.096,A -85,B 0,C 180,E1 -18255.472,E2 -18255.472} C_VEL
LIN {X 0,Y 261.776,Z 368.694,A -85,B 0,C 180,E1 -18257.598,E2 -18257.598} C_VEL
LIN {X 0,Y 262.362,Z 363.752,A -85,B 0,C 180,E1 -18259.973,E2 -18259.973} C_VEL
LIN {X 0,Y 263.294,Z 357.487,A -85,B 0,C 180,E1 -18262.33,E2 -18262.33} C_VEL
LIN {X 0,Y 264.423,Z 349.705,A -85,B 0,C 180,E1 -18264.663,E2 -18264.663} C_VEL
LIN {X 0,Y 265.664,Z 341.691,A -85,B 0,C 180,E1 -18266.588,E2 -18266.588} C_VEL
LIN {X 0,Y 267.197,Z 331.864,A -85,B 0,C 180,E1 -18268.493,E2 -18268.493} C_VEL
LIN {X 0,Y 268.648,Z 320.984,A -85,B 0,C 180,E1 -18270.188,E2 -18270.188} C_VEL
LIN {X 0,Y 269.981,Z 310.372,A -85,B 0,C 180,E1 -18271.492,E2 -18271.492} C_VEL
LIN {X 0,Y 271.147,Z 297.686,A -85,B 0,C 180,E1 -18272.693,E2 -18272.693} C_VEL
LIN {X 0,Y 272.055,Z 285.038,A -85,B 0,C 180,E1 -18273.564,E2 -18273.564} C_VEL
LIN {X 0,Y 272.748,Z 273.023,A -85,B 0,C 180,E1 -18274.11,E2 -18274.11} C_VEL
LIN {X 0,Y 274.824,Z 199.612,A -85,B 0,C 180,E1 -18276.05,E2 -18276.05} C_VEL
LIN {X 0,Y 272.976,Z 192.315,A -85,B 0,C 180,E1 -18276.404,E2 -18276.404} C_VEL
LIN {X 0,Y 264.308,Z 168.36,A -85,B 0,C 180,E1 -18277.84,E2 -18277.84} C_VEL
LIN {X 0,Y 263.622,Z 166.359,A -85,B 0,C 180,E1 -18278,E2 -18278} C_VEL
LIN {X 0,Y 263.498,Z 165.665,A -85,B 0,C 180,E1 -18278.343,E2 -18278.343} C_VEL
LIN {X 0,Y 263.285,Z 165.69,A -85,B 0,C 180,E1 -18282.331,E2 -18282.331} C_VEL
LIN {X 0,Y 263.249,Z 165.695,A -85,B 0,C 180,E1 -18286.038,E2 -18286.038} C_VEL
LIN {X 0,Y 263.168,Z 165.702,A -85,B 0,C 180,E1 -18290.825,E2 -18290.825} C_VEL
LIN {X 0,Y 263.1,Z 165.688,A -85,B 0,C 180,E1 -18295.303,E2 -18295.303} C_VEL
LIN {X 0,Y 263.114,Z 165.701,A -85,B 0,C 180,E1 -18298.738,E2 -18298.738} C_VEL
LIN {X 0,Y 263.124,Z 165.707,A -85,B 0,C 180,E1 -18302.29,E2 -18302.29} C_VEL
LIN {X 0,Y 263.173,Z 165.692,A -85,B 0,C 180,E1 -18306.762,E2 -18306.762} C_VEL
LIN {X 0,Y 263.089,Z 165.711,A -85,B 0,C 180,E1 -18309.876,E2 -18309.876} C_VEL
LIN {X 0,Y 263.074,Z 165.708,A -85,B 0,C 180,E1 -18313.995,E2 -18313.995} C_VEL
LIN {X 0,Y 263.079,Z 165.702,A -85,B 0,C 180,E1 -18318.419,E2 -18318.419} C_VEL
LIN {X 0,Y 263.156,Z 165.702,A -85,B 0,C 180,E1 -18322.104,E2 -18322.104} C_VEL
LIN {X 0,Y 263.151,Z 165.7,A -85,B 0,C 180,E1 -18325.887,E2 -18325.887} C_VEL
LIN {X 0,Y 263.109,Z 165.69,A -85,B 0,C 180,E1 -18329.503,E2 -18329.503} C_VEL
LIN {X 0,Y 263.113,Z 165.701,A -85,B 0,C 180,E1 -18332.995,E2 -18332.995} C_VEL
LIN {X 0,Y 263.116,Z 165.709,A -85,B 0,C 180,E1 -18336.382,E2 -18336.382} C_VEL
LIN {X 0,Y 263.208,Z 165.697,A -85,B 0,C 180,E1 -18339.69,E2 -18339.69} C_VEL
LIN {X 0,Y 263.29,Z 165.688,A -85,B 0,C 180,E1 -18344.519,E2 -18344.519} C_VEL
LIN {X 0,Y 263.33,Z 165.68,A -85,B 0,C 180,E1 -18349.233,E2 -18349.233} C_VEL
LIN {X 0,Y 263.53,Z 165.657,A -85,B 0,C 180,E1 -18352.338,E2 -18352.338} C_VEL
LIN {X 0,Y 263.39,Z 165.673,A -85,B 0,C 180,E1 -18354.618,E2 -18354.618} C_VEL
LIN {X 0,Y 262.671,Z 165.768,A -85,B 0,C 180,E1 -18355.897,E2 -18355.897} C_VEL
LIN {X 0,Y 259.923,Z 166.106,A -85,B 0,C 180,E1 -18357.986,E2 -18357.986} C_VEL
LIN {X 0,Y 257.669,Z 166.384,A -85,B 0,C 180,E1 -18359.685,E2 -18359.685} C_VEL
LIN {X 0,Y 256.747,Z 166.498,A -85,B 0,C 180,E1 -18360.998,E2 -18360.998} C_VEL
LIN {X 0,Y 256.692,Z 166.507,A -85,B 0,C 180,E1 -18361.442,E2 -18361.442} C_VEL
LIN {X 0,Y 256.457,Z 166.536,A -85,B 0,C 180,E1 -18366.294,E2 -18366.294} C_VEL
LIN {X 0,Y 256.431,Z 166.539,A -85,B 0,C 180,E1 -18369.466,E2 -18369.466} C_VEL
LIN {X 0,Y 256.211,Z 166.567,A -85,B 0,C 180,E1 -18374.293,E2 -18374.293} C_VEL
LIN {X 0,Y 256.153,Z 166.576,A -85,B 0,C 180,E1 -18377.567,E2 -18377.567} C_VEL
LIN {X 0,Y 256.126,Z 166.582,A -85,B 0,C 180,E1 -18381.099,E2 -18381.099} C_VEL
LIN {X 0,Y 256.137,Z 166.58,A -85,B 0,C 180,E1 -18385.112,E2 -18385.112} C_VEL
LIN {X 0,Y 256.059,Z 166.588,A -85,B 0,C 180,E1 -18389.608,E2 -18389.608} C_VEL
LIN {X 0,Y 256.07,Z 166.589,A -85,B 0,C 180,E1 -18393.293,E2 -18393.293} C_VEL
LIN {X 0,Y 256.116,Z 166.583,A -85,B 0,C 180,E1 -18397.27,E2 -18397.27} C_VEL
LIN {X 0,Y 256.023,Z 166.596,A -85,B 0,C 180,E1 -18401.211,E2 -18401.211} C_VEL
LIN {X 0,Y 256.021,Z 166.595,A -85,B 0,C 180,E1 -18405.54,E2 -18405.54} C_VEL
LIN {X 0,Y 256.044,Z 166.593,A -85,B 0,C 180,E1 -18408.794,E2 -18408.794} C_VEL
LIN {X 0,Y 256.13,Z 166.58,A -85,B 0,C 180,E1 -18412.867,E2 -18412.867} C_VEL
LIN {X 0,Y 256.119,Z 166.737,A -85,B 0,C 180,E1 -18415.697,E2 -18415.697} C_VEL
LIN {X 0,Y 258.263,Z 176.687,A -85,B 0,C 180,E1 -18419.267,E2 -18419.267} C_VEL
LIN {X 0,Y 259.639,Z 183.677,A -85,B 0,C 180,E1 -18421.672,E2 -18421.672} C_VEL
LIN {X 0,Y 262.383,Z 192.486,A -85,B 0,C 180,E1 -18422.197,E2 -18422.197} C_VEL
LIN {X 0,Y 267.448,Z 232.613,A -85,B 0,C 180,E1 -18423.798,E2 -18423.798} C_VEL
LIN {X 0,Y 265.684,Z 292.4,A -85,B 0,C 180,E1 -18425.43,E2 -18425.43} C_VEL
LIN {X 0,Y 264.85,Z 305.601,A -85,B 0,C 180,E1 -18426.077,E2 -18426.077} C_VEL
LIN {X 0,Y 263.547,Z 318.871,A -85,B 0,C 180,E1 -18427.045,E2 -18427.045} C_VEL
LIN {X 0,Y 262.223,Z 330.05,A -85,B 0,C 180,E1 -18428.168,E2 -18428.168} C_VEL
LIN {X 0,Y 260.514,Z 341.681,A -85,B 0,C 180,E1 -18429.675,E2 -18429.675} C_VEL
LIN {X 0,Y 259.039,Z 352.411,A -85,B 0,C 180,E1 -18431.451,E2 -18431.451} C_VEL
LIN {X 0,Y 257.885,Z 359.863,A -85,B 0,C 180,E1 -18432.964,E2 -18432.964} C_VEL
LIN {X 0,Y 256.666,Z 367.913,A -85,B 0,C 180,E1 -18434.922,E2 -18434.922} C_VEL
LIN {X 0,Y 255.444,Z 375.751,A -85,B 0,C 180,E1 -18437.285,E2 -18437.285} C_VEL
LIN {X 0,Y 254.722,Z 382.025,A -85,B 0,C 180,E1 -18439.668,E2 -18439.668} C_VEL
LIN {X 0,Y 254.29,Z 386.989,A -85,B 0,C 180,E1 -18442.057,E2 -18442.057} C_VEL
LIN {X 0,Y 254.056,Z 391.273,A -85,B 0,C 180,E1 -18444.801,E2 -18444.801} C_VEL
LIN {X 0,Y 254.071,Z 393.547,A -85,B 0,C 180,E1 -18446.828,E2 -18446.828} C_VEL
LIN {X 0,Y 254.093,Z 394.833,A -85,B 0,C 180,E1 -18448.415,E2 -18448.415} C_VEL
LIN {X 0,Y 254.103,Z 395.715,A -85,B 0,C 180,E1 -18450,E2 -18450} C_VEL
LIN {X 0,Y 254.068,Z 396.173,A -85,B 0,C 180,E1 -18451.585,E2 -18451.585} C_VEL
LIN {X 0,Y 254.016,Z 396.209,A -85,B 0,C 180,E1 -18453.172,E2 -18453.172} C_VEL
LIN {X 0,Y 254.061,Z 395.132,A -85,B 0,C 180,E1 -18456.353,E2 -18456.353} C_VEL
LIN {X 0,Y 254.272,Z 394.01,A -85,B 0,C 180,E1 -18457.943,E2 -18457.943} C_VEL
LIN {X 0,Y 254.663,Z 392.448,A -85,B 0,C 180,E1 -18459.531,E2 -18459.531} C_VEL
LIN {X 0,Y 255.491,Z 389.342,A -85,B 0,C 180,E1 -18461.906,E2 -18461.906} C_VEL
LIN {X 0,Y 256.694,Z 385.209,A -85,B 0,C 180,E1 -18464.265,E2 -18464.265} C_VEL
LIN {X 0,Y 258.852,Z 378.924,A -85,B 0,C 180,E1 -18466.97,E2 -18466.97} C_VEL
LIN {X 0,Y 260.771,Z 372.363,A -85,B 0,C 180,E1 -18469.199,E2 -18469.199} C_VEL
LIN {X 0,Y 262.961,Z 365.219,A -85,B 0,C 180,E1 -18471.15,E2 -18471.15} C_VEL
LIN {X 0,Y 265.425,Z 356.932,A -85,B 0,C 180,E1 -18472.989,E2 -18472.989} C_VEL
LIN {X 0,Y 268.219,Z 346.8,A -85,B 0,C 180,E1 -18474.787,E2 -18474.787} C_VEL
LIN {X 0,Y 270.907,Z 335.399,A -85,B 0,C 180,E1 -18476.376,E2 -18476.376} C_VEL
LIN {X 0,Y 273.275,Z 324.214,A -85,B 0,C 180,E1 -18477.576,E2 -18477.576} C_VEL
LIN {X 0,Y 275.459,Z 311.634,A -85,B 0,C 180,E1 -18478.58,E2 -18478.58} C_VEL
LIN {X 0,Y 277.112,Z 298.803,A -85,B 0,C 180,E1 -18479.296,E2 -18479.296} C_VEL
LIN {X 0,Y 278.043,Z 285.975,A -85,B 0,C 180,E1 -18479.766,E2 -18479.766} C_VEL
LIN {X 0,Y 280,Z 236.195,A -85,B 0,C 180,E1 -18481.079,E2 -18481.079} C_VEL
LIN {X 0,Y 277.142,Z 217.862,A -85,B 0,C 180,E1 -18482.132,E2 -18482.132} C_VEL
LIN {X 0,Y 276.209,Z 213.578,A -85,B 0,C 180,E1 -18482.429,E2 -18482.429} C_VEL
LIN {X 0,Y 269.874,Z 199.636,A -85,B 0,C 180,E1 -18483.993,E2 -18483.993} C_VEL
LIN {X 0,Y 264.634,Z 189.79,A -85,B 0,C 180,E1 -18485.31,E2 -18485.31} C_VEL
LIN {X 0,Y 262.481,Z 185.835,A -85,B 0,C 180,E1 -18485.872,E2 -18485.872} C_VEL
LIN {X 0,Y 260.447,Z 181.87,A -85,B 0,C 180,E1 -18486.432,E2 -18486.432} C_VEL
LIN {X 0,Y 258.111,Z 173.512,A -85,B 0,C 180,E1 -18490.323,E2 -18490.323} C_VEL
LIN {X 0,Y 256.047,Z 166.589,A -85,B 0,C 180,E1 -18493.943,E2 -18493.943} C_VEL
LIN {X 0,Y 256.057,Z 166.591,A -85,B 0,C 180,E1 -18497.823,E2 -18497.823} C_VEL
LIN {X 0,Y 256.067,Z 166.589,A -85,B 0,C 180,E1 -18500.856,E2 -18500.856} C_VEL
LIN {X 0,Y 256.082,Z 166.58,A -85,B 0,C 180,E1 -18504.806,E2 -18504.806} C_VEL
LIN {X 0,Y 256.085,Z 166.577,A -85,B 0,C 180,E1 -18508.57,E2 -18508.57} C_VEL
LIN {X 0,Y 256.083,Z 166.577,A -85,B 0,C 180,E1 -18512.188,E2 -18512.188} C_VEL
LIN {X 0,Y 256.088,Z 166.584,A -85,B 0,C 180,E1 -18515.69,E2 -18515.69} C_VEL
LIN {X 0,Y 256.123,Z 166.578,A -85,B 0,C 180,E1 -18519.1,E2 -18519.1} C_VEL
LIN {X 0,Y 256.215,Z 166.569,A -85,B 0,C 180,E1 -18524.079,E2 -18524.079} C_VEL
LIN {X 0,Y 256.276,Z 166.561,A -85,B 0,C 180,E1 -18528.932,E2 -18528.932} C_VEL
LIN {X 0,Y 256.47,Z 166.523,A -85,B 0,C 180,E1 -18532.124,E2 -18532.124} C_VEL
LIN {X 0,Y 256.453,Z 166.523,A -85,B 0,C 180,E1 -18536.857,E2 -18536.857} C_VEL
LIN {X 0,Y 256.701,Z 166.506,A -85,B 0,C 180,E1 -18538.43,E2 -18538.43} C_VEL
LIN {X 0,Y 256.708,Z 166.493,A -85,B 0,C 180,E1 -18541.568,E2 -18541.568} C_VEL
LIN {X 0,Y 256.451,Z 166.528,A -85,B 0,C 180,E1 -18546.566,E2 -18546.566} C_VEL
LIN {X 0,Y 256.428,Z 166.535,A -85,B 0,C 180,E1 -18549.464,E2 -18549.464} C_VEL
LIN {X 0,Y 256.238,Z 166.557,A -85,B 0,C 180,E1 -18554.29,E2 -18554.29} C_VEL
LIN {X 0,Y 256.182,Z 166.568,A -85,B 0,C 180,E1 -18557.563,E2 -18557.563} C_VEL
LIN {X 0,Y 256.15,Z 166.574,A -85,B 0,C 180,E1 -18561.114,E2 -18561.114} C_VEL
LIN {X 0,Y 256.171,Z 166.571,A -85,B 0,C 180,E1 -18565.129,E2 -18565.129} C_VEL
LIN {X 0,Y 256.113,Z 166.585,A -85,B 0,C 180,E1 -18569.599,E2 -18569.599} C_VEL
LIN {X 0,Y 256.102,Z 166.658,A -85,B 0,C 180,E1 -18571.828,E2 -18571.828} C_VEL
LIN {X 0,Y 256.71,Z 168.672,A -85,B 0,C 180,E1 -18572.818,E2 -18572.818} C_VEL
LIN {X 0,Y 259.419,Z 172.826,A -85,B 0,C 180,E1 -18573.56,E2 -18573.56} C_VEL
LIN {X 0,Y 267.579,Z 186.191,A -85,B 0,C 180,E1 -18575.662,E2 -18575.662} C_VEL
LIN {X 0,Y 275.297,Z 200.634,A -85,B 0,C 180,E1 -18577.531,E2 -18577.531} C_VEL
LIN {X 0,Y 280.956,Z 213.132,A -85,B 0,C 180,E1 -18578.869,E2 -18578.869} C_VEL
LIN {X 0,Y 278.257,Z 275.509,A -85,B 0,C 180,E1 -18580.532,E2 -18580.532} C_VEL
LIN {X 0,Y 276.989,Z 288.839,A -85,B 0,C 180,E1 -18581.158,E2 -18581.158} C_VEL
LIN {X 0,Y 275.449,Z 301.774,A -85,B 0,C 180,E1 -18582.1,E2 -18582.1} C_VEL
LIN {X 0,Y 273.456,Z 312.963,A -85,B 0,C 180,E1 -18583.176,E2 -18583.176} C_VEL
LIN {X 0,Y 271.259,Z 323.617,A -85,B 0,C 180,E1 -18584.504,E2 -18584.504} C_VEL
LIN {X 0,Y 268.717,Z 333.98,A -85,B 0,C 180,E1 -18586.126,E2 -18586.126} C_VEL
LIN {X 0,Y 266.16,Z 343.273,A -85,B 0,C 180,E1 -18587.954,E2 -18587.954} C_VEL
LIN {X 0,Y 263.398,Z 352.21,A -85,B 0,C 180,E1 -18590.181,E2 -18590.181} C_VEL
LIN {X 0,Y 260.869,Z 360.072,A -85,B 0,C 180,E1 -18592.687,E2 -18592.687} C_VEL
LIN {X 0,Y 258.746,Z 366.162,A -85,B 0,C 180,E1 -18595.222,E2 -18595.222} C_VEL
LIN {X 0,Y 256.946,Z 371.137,A -85,B 0,C 180,E1 -18597.984,E2 -18597.984} C_VEL
LIN {X 0,Y 255.763,Z 374.228,A -85,B 0,C 180,E1 -18600.356,E2 -18600.356} C_VEL
LIN {X 0,Y 255.096,Z 375.872,A -85,B 0,C 180,E1 -18602.072,E2 -18602.072} C_VEL
LIN {X 0,Y 254.592,Z 376.99,A -85,B 0,C 180,E1 -18603.789,E2 -18603.789} C_VEL
LIN {X 0,Y 254.199,Z 377.744,A -85,B 0,C 180,E1 -18605.833,E2 -18605.833} C_VEL
LIN {X 0,Y 253.828,Z 377.63,A -85,B 0,C 180,E1 -18608.903,E2 -18608.903} C_VEL
LIN {X 0,Y 253.829,Z 376.937,A -85,B 0,C 180,E1 -18610.594,E2 -18610.594} C_VEL
LIN {X 0,Y 253.84,Z 375.833,A -85,B 0,C 180,E1 -18612.269,E2 -18612.269} C_VEL
LIN {X 0,Y 254.012,Z 374.239,A -85,B 0,C 180,E1 -18613.938,E2 -18613.938} C_VEL
LIN {X 0,Y 254.439,Z 370.996,A -85,B 0,C 180,E1 -18616.421,E2 -18616.421} C_VEL
LIN {X 0,Y 254.966,Z 366.648,A -85,B 0,C 180,E1 -18618.875,E2 -18618.875} C_VEL
LIN {X 0,Y 255.823,Z 360.607,A -85,B 0,C 180,E1 -18621.485,E2 -18621.485} C_VEL
LIN {X 0,Y 256.807,Z 354.081,A -85,B 0,C 180,E1 -18623.716,E2 -18623.716} C_VEL
LIN {X 0,Y 257.947,Z 346.934,A -85,B 0,C 180,E1 -18625.703,E2 -18625.703} C_VEL
LIN {X 0,Y 259.3,Z 338.304,A -85,B 0,C 180,E1 -18627.67,E2 -18627.67} C_VEL
LIN {X 0,Y 260.864,Z 328.242,A -85,B 0,C 180,E1 -18629.507,E2 -18629.507} C_VEL
LIN {X 0,Y 262.337,Z 316.979,A -85,B 0,C 180,E1 -18631.152,E2 -18631.152} C_VEL
LIN {X 0,Y 263.701,Z 305.263,A -85,B 0,C 180,E1 -18632.482,E2 -18632.482} C_VEL
LIN {X 0,Y 264.813,Z 293.094,A -85,B 0,C 180,E1 -18633.519,E2 -18633.519} C_VEL
LIN {X 0,Y 265.64,Z 279.966,A -85,B 0,C 180,E1 -18634.315,E2 -18634.315} C_VEL
LIN {X 0,Y 266.225,Z 267.278,A -85,B 0,C 180,E1 -18634.78,E2 -18634.78} C_VEL
LIN {X 0,Y 268.183,Z 200.517,A -85,B 0,C 180,E1 -18636.561,E2 -18636.561} C_VEL
LIN {X 0,Y 265.938,Z 192.731,A -85,B 0,C 180,E1 -18636.977,E2 -18636.977} C_VEL
LIN {X 0,Y 258.336,Z 171.583,A -85,B 0,C 180,E1 -18638.291,E2 -18638.291} C_VEL
LIN {X 0,Y 256.489,Z 166.748,A -85,B 0,C 180,E1 -18638.619,E2 -18638.619} C_VEL
LIN {X 0,Y 256.267,Z 166.564,A -85,B 0,C 180,E1 -18641.068,E2 -18641.068} C_VEL
LIN {X 0,Y 256.209,Z 166.573,A -85,B 0,C 180,E1 -18645.921,E2 -18645.921} C_VEL
LIN {X 0,Y 256.114,Z 166.582,A -85,B 0,C 180,E1 -18651.097,E2 -18651.097} C_VEL
LIN {X 0,Y 256.073,Z 166.561,A -85,B 0,C 180,E1 -18655.085,E2 -18655.085} C_VEL
LIN {X 0,Y 256.073,Z 166.577,A -85,B 0,C 180,E1 -18658.57,E2 -18658.57} C_VEL
LIN {X 0,Y 256.067,Z 166.588,A -85,B 0,C 180,E1 -18661.7,E2 -18661.7} C_VEL
LIN {X 0,Y 256.077,Z 166.578,A -85,B 0,C 180,E1 -18665.194,E2 -18665.194} C_VEL
LIN {X 0,Y 256.108,Z 166.575,A -85,B 0,C 180,E1 -18667.27,E2 -18667.27} C_VEL
LIN {X 0,Y 256.016,Z 166.595,A -85,B 0,C 180,E1 -18671.212,E2 -18671.212} C_VEL
LIN {X 0,Y 256.016,Z 166.579,A -85,B 0,C 180,E1 -18675.541,E2 -18675.541} C_VEL
LIN {X 0,Y 256.017,Z 166.584,A -85,B 0,C 180,E1 -18678.79,E2 -18678.79} C_VEL
LIN {X 0,Y 256.125,Z 166.582,A -85,B 0,C 180,E1 -18682.868,E2 -18682.868} C_VEL
LIN {X 0,Y 256.065,Z 166.58,A -85,B 0,C 180,E1 -18686.708,E2 -18686.708} C_VEL
LIN {X 0,Y 256.041,Z 166.568,A -85,B 0,C 180,E1 -18690.392,E2 -18690.392} C_VEL
LIN {X 0,Y 256.066,Z 166.577,A -85,B 0,C 180,E1 -18693.952,E2 -18693.952} C_VEL
LIN {X 0,Y 256.058,Z 166.587,A -85,B 0,C 180,E1 -18697.403,E2 -18697.403} C_VEL
LIN {X 0,Y 256.104,Z 166.58,A -85,B 0,C 180,E1 -18700.774,E2 -18700.774} C_VEL
LIN {X 0,Y 256.215,Z 166.566,A -85,B 0,C 180,E1 -18704.081,E2 -18704.081} C_VEL
LIN {X 0,Y 256.273,Z 166.559,A -85,B 0,C 180,E1 -18708.933,E2 -18708.933} C_VEL
LIN {X 0,Y 256.472,Z 166.534,A -85,B 0,C 180,E1 -18712.126,E2 -18712.126} C_VEL
LIN {X 0,Y 256.448,Z 166.539,A -85,B 0,C 180,E1 -18716.859,E2 -18716.859} C_VEL
LIN {X 0,Y 256.697,Z 166.505,A -85,B 0,C 180,E1 -18718.432,E2 -18718.432} C_VEL
LIN {X 0,Y 256.692,Z 166.507,A -85,B 0,C 180,E1 -18721.442,E2 -18721.442} C_VEL
LIN {X 0,Y 256.061,Z 166.592,A -85,B 0,C 180,E1 -18722.748,E2 -18722.748} C_VEL
LIN {X 0,Y 253.153,Z 166.956,A -85,B 0,C 180,E1 -18724.874,E2 -18724.874} C_VEL
LIN {X 0,Y 250.627,Z 167.265,A -85,B 0,C 180,E1 -18726.604,E2 -18726.604} C_VEL
LIN {X 0,Y 249.509,Z 167.4,A -85,B 0,C 180,E1 -18727.948,E2 -18727.948} C_VEL
LIN {X 0,Y 249.402,Z 167.412,A -85,B 0,C 180,E1 -18728.405,E2 -18728.405} C_VEL
LIN {X 0,Y 249.179,Z 167.446,A -85,B 0,C 180,E1 -18733.041,E2 -18733.041} C_VEL
LIN {X 0,Y 249.155,Z 167.442,A -85,B 0,C 180,E1 -18736.451,E2 -18736.451} C_VEL
LIN {X 0,Y 249.05,Z 167.462,A -85,B 0,C 180,E1 -18741.522,E2 -18741.522} C_VEL
LIN {X 0,Y 249.089,Z 167.458,A -85,B 0,C 180,E1 -18745.46,E2 -18745.46} C_VEL
LIN {X 0,Y 249.041,Z 167.464,A -85,B 0,C 180,E1 -18748.974,E2 -18748.974} C_VEL
LIN {X 0,Y 249.032,Z 167.463,A -85,B 0,C 180,E1 -18752.427,E2 -18752.427} C_VEL
LIN {X 0,Y 249.032,Z 167.464,A -85,B 0,C 180,E1 -18756.346,E2 -18756.346} C_VEL
LIN {X 0,Y 248.983,Z 167.473,A -85,B 0,C 180,E1 -18760.484,E2 -18760.484} C_VEL
LIN {X 0,Y 248.966,Z 167.476,A -85,B 0,C 180,E1 -18764.889,E2 -18764.889} C_VEL
LIN {X 0,Y 248.997,Z 167.469,A -85,B 0,C 180,E1 -18767.358,E2 -18767.358} C_VEL
LIN {X 0,Y 249.044,Z 167.461,A -85,B 0,C 180,E1 -18772.201,E2 -18772.201} C_VEL
LIN {X 0,Y 249.059,Z 167.465,A -85,B 0,C 180,E1 -18775.174,E2 -18775.174} C_VEL
LIN {X 0,Y 251.148,Z 177.336,A -85,B 0,C 180,E1 -18778.822,E2 -18778.822} C_VEL
LIN {X 0,Y 252.455,Z 183.704,A -85,B 0,C 180,E1 -18781.018,E2 -18781.018} C_VEL
LIN {X 0,Y 255.981,Z 194.702,A -85,B 0,C 180,E1 -18781.69,E2 -18781.69} C_VEL
LIN {X 0,Y 260.786,Z 233.51,A -85,B 0,C 180,E1 -18783.285,E2 -18783.285} C_VEL
LIN {X 0,Y 259.007,Z 291.886,A -85,B 0,C 180,E1 -18784.914,E2 -18784.914} C_VEL
LIN {X 0,Y 258.143,Z 305.17,A -85,B 0,C 180,E1 -18785.576,E2 -18785.576} C_VEL
LIN {X 0,Y 256.876,Z 317.936,A -85,B 0,C 180,E1 -18786.52,E2 -18786.52} C_VEL
LIN {X 0,Y 255.384,Z 330.102,A -85,B 0,C 180,E1 -18787.765,E2 -18787.765} C_VEL
LIN {X 0,Y 253.62,Z 341.675,A -85,B 0,C 180,E1 -18789.31,E2 -18789.31} C_VEL
LIN {X 0,Y 252.139,Z 352.151,A -85,B 0,C 180,E1 -18791.093,E2 -18791.093} C_VEL
LIN {X 0,Y 250.79,Z 360.712,A -85,B 0,C 180,E1 -18792.896,E2 -18792.896} C_VEL
LIN {X 0,Y 249.361,Z 369.902,A -85,B 0,C 180,E1 -18795.306,E2 -18795.306} C_VEL
LIN {X 0,Y 248.156,Z 377.302,A -85,B 0,C 180,E1 -18797.736,E2 -18797.736} C_VEL
LIN {X 0,Y 247.519,Z 383.236,A -85,B 0,C 180,E1 -18800.191,E2 -18800.191} C_VEL
LIN {X 0,Y 247.114,Z 387.88,A -85,B 0,C 180,E1 -18802.647,E2 -18802.647} C_VEL
LIN {X 0,Y 246.933,Z 391.388,A -85,B 0,C 180,E1 -18805.102,E2 -18805.102} C_VEL
LIN {X 0,Y 246.984,Z 393.142,A -85,B 0,C 180,E1 -18806.737,E2 -18806.737} C_VEL
LIN {X 0,Y 247.021,Z 394.461,A -85,B 0,C 180,E1 -18808.369,E2 -18808.369} C_VEL
LIN {X 0,Y 247.03,Z 395.375,A -85,B 0,C 180,E1 -18810,E2 -18810} C_VEL
LIN {X 0,Y 246.996,Z 395.888,A -85,B 0,C 180,E1 -18811.63,E2 -18811.63} C_VEL
LIN {X 0,Y 246.913,Z 395.963,A -85,B 0,C 180,E1 -18813.263,E2 -18813.263} C_VEL
LIN {X 0,Y 246.916,Z 395.621,A -85,B 0,C 180,E1 -18814.981,E2 -18814.981} C_VEL
LIN {X 0,Y 247.214,Z 393.872,A -85,B 0,C 180,E1 -18818.172,E2 -18818.172} C_VEL
LIN {X 0,Y 247.637,Z 392.364,A -85,B 0,C 180,E1 -18819.804,E2 -18819.804} C_VEL
LIN {X 0,Y 248.525,Z 389.327,A -85,B 0,C 180,E1 -18822.245,E2 -18822.245} C_VEL
LIN {X 0,Y 249.82,Z 385.265,A -85,B 0,C 180,E1 -18824.666,E2 -18824.666} C_VEL
LIN {X 0,Y 252.047,Z 379.063,A -85,B 0,C 180,E1 -18827.442,E2 -18827.442} C_VEL
LIN {X 0,Y 254.398,Z 371.517,A -85,B 0,C 180,E1 -18830.066,E2 -18830.066} C_VEL
LIN {X 0,Y 256.829,Z 364.062,A -85,B 0,C 180,E1 -18832.102,E2 -18832.102} C_VEL
LIN {X 0,Y 259.499,Z 355.571,A -85,B 0,C 180,E1 -18833.969,E2 -18833.969} C_VEL
LIN {X 0,Y 262.395,Z 345.134,A -85,B 0,C 180,E1 -18835.801,E2 -18835.801} C_VEL
LIN {X 0,Y 264.971,Z 334.841,A -85,B 0,C 180,E1 -18837.228,E2 -18837.228} C_VEL
LIN {X 0,Y 267.422,Z 323.612,A -85,B 0,C 180,E1 -18838.446,E2 -18838.446} C_VEL
LIN {X 0,Y 269.684,Z 310.91,A -85,B 0,C 180,E1 -18839.465,E2 -18839.465} C_VEL
LIN {X 0,Y 271.369,Z 298.293,A -85,B 0,C 180,E1 -18840.171,E2 -18840.171} C_VEL
LIN {X 0,Y 272.329,Z 285.344,A -85,B 0,C 180,E1 -18840.649,E2 -18840.649} C_VEL
LIN {X 0,Y 274.3,Z 236.941,A -85,B 0,C 180,E1 -18841.955,E2 -18841.955} C_VEL
LIN {X 0,Y 271.26,Z 217.405,A -85,B 0,C 180,E1 -18843.13,E2 -18843.13} C_VEL
LIN {X 0,Y 265.294,Z 204.051,A -85,B 0,C 180,E1 -18844.668,E2 -18844.668} C_VEL
LIN {X 0,Y 258.428,Z 190.949,A -85,B 0,C 180,E1 -18846.494,E2 -18846.494} C_VEL
LIN {X 0,Y 255.283,Z 185.544,A -85,B 0,C 180,E1 -18847.371,E2 -18847.371} C_VEL
LIN {X 0,Y 253.059,Z 181.424,A -85,B 0,C 180,E1 -18848.052,E2 -18848.052} C_VEL
LIN {X 0,Y 251.38,Z 175.426,A -85,B 0,C 180,E1 -18850.986,E2 -18850.986} C_VEL
LIN {X 0,Y 248.984,Z 167.474,A -85,B 0,C 180,E1 -18855.328,E2 -18855.328} C_VEL
LIN {X 0,Y 248.984,Z 167.466,A -85,B 0,C 180,E1 -18859.652,E2 -18859.652} C_VEL
LIN {X 0,Y 249.043,Z 167.464,A -85,B 0,C 180,E1 -18863.656,E2 -18863.656} C_VEL
LIN {X 0,Y 249.035,Z 167.461,A -85,B 0,C 180,E1 -18867.847,E2 -18867.847} C_VEL
LIN {X 0,Y 249.046,Z 167.461,A -85,B 0,C 180,E1 -18871.331,E2 -18871.331} C_VEL
LIN {X 0,Y 249.058,Z 167.46,A -85,B 0,C 180,E1 -18874.958,E2 -18874.958} C_VEL
